LIN {X 0,Y 435.105,Z 1048.847,A -85,B 0,C 180,E1 20642.919,E2 20642.919} C_VEL
LIN {X 0,Y 432.049,Z 1065.311,A -85,B 0,C 180,E1 20641.068,E2 20641.068} C_VEL
LIN {X 0,Y 428.929,Z 1081.421,A -85,B 0,C 180,E1 20638.926,E2 20638.926} C_VEL
LIN {X 0,Y 426.223,Z 1095.243,A -85,B 0,C 180,E1 20636.769,E2 20636.769} C_VEL
LIN {X 0,Y 423.614,Z 1108.344,A -85,B 0,C 180,E1 20634.345,E2 20634.345} C_VEL
LIN {X 0,Y 421.322,Z 1120.264,A -85,B 0,C 180,E1 20631.728,E2 20631.728} C_VEL
LIN {X 0,Y 419.538,Z 1130.485,A -85,B 0,C 180,E1 20629.056,E2 20629.056} C_VEL
LIN {X 0,Y 418.131,Z 1139.349,A -85,B 0,C 180,E1 20626.246,E2 20626.246} C_VEL
LIN {X 0,Y 417.148,Z 1146.8,A -85,B 0,C 180,E1 20623.303,E2 20623.303} C_VEL
LIN {X 0,Y 416.528,Z 1152.908,A -85,B 0,C 180,E1 20620.201,E2 20620.201} C_VEL
LIN {X 0,Y 416.233,Z 1157.103,A -85,B 0,C 180,E1 20617.314,E2 20617.314} C_VEL
LIN {X 0,Y 416.088,Z 1159.912,A -85,B 0,C 180,E1 20614.272,E2 20614.272} C_VEL
LIN {X 0,Y 416.05,Z 1161.297,A -85,B 0,C 180,E1 20611.102,E2 20611.102} C_VEL
LIN {X 0,Y 416.047,Z 1161.219,A -85,B 0,C 180,E1 20608.21,E2 20608.21} C_VEL
LIN {X 0,Y 416.098,Z 1159.578,A -85,B 0,C 180,E1 20605.176,E2 20605.176} C_VEL
LIN {X 0,Y 416.291,Z 1156.297,A -85,B 0,C 180,E1 20601.993,E2 20601.993} C_VEL
LIN {X 0,Y 416.638,Z 1151.851,A -85,B 0,C 180,E1 20599.072,E2 20599.072} C_VEL
LIN {X 0,Y 417.28,Z 1145.733,A -85,B 0,C 180,E1 20596.137,E2 20596.137} C_VEL
LIN {X 0,Y 418.332,Z 1137.948,A -85,B 0,C 180,E1 20593.19,E2 20593.19} C_VEL
LIN {X 0,Y 419.837,Z 1128.815,A -85,B 0,C 180,E1 20590.38,E2 20590.38} C_VEL
LIN {X 0,Y 421.711,Z 1118.284,A -85,B 0,C 180,E1 20587.707,E2 20587.707} C_VEL
LIN {X 0,Y 423.979,Z 1106.39,A -85,B 0,C 180,E1 20585.181,E2 20585.181} C_VEL
LIN {X 0,Y 426.622,Z 1093.222,A -85,B 0,C 180,E1 20582.806,E2 20582.806} C_VEL
LIN {X 0,Y 429.496,Z 1078.65,A -85,B 0,C 180,E1 20580.581,E2 20580.581} C_VEL
LIN {X 0,Y 432.519,Z 1062.81,A -85,B 0,C 180,E1 20578.542,E2 20578.542} C_VEL
LIN {X 0,Y 435.66,Z 1045.506,A -85,B 0,C 180,E1 20576.657,E2 20576.657} C_VEL
LIN {X 0,Y 438.639,Z 1027.657,A -85,B 0,C 180,E1 20575.022,E2 20575.022} C_VEL
LIN {X 0,Y 441.258,Z 1009.727,A -85,B 0,C 180,E1 20573.664,E2 20573.664} C_VEL
LIN {X 0,Y 443.774,Z 989.808,A -85,B 0,C 180,E1 20572.414,E2 20572.414} C_VEL
LIN {X 0,Y 445.795,Z 970.199,A -85,B 0,C 180,E1 20571.428,E2 20571.428} C_VEL
LIN {X 0,Y 447.419,Z 949.171,A -85,B 0,C 180,E1 20570.621,E2 20570.621} C_VEL
LIN {X 0,Y 448.598,Z 926.606,A -85,B 0,C 180,E1 20570.002,E2 20570.002} C_VEL
LIN {X 0,Y 454.402,Z 736.319,A -85,B 0,C 180,E1 20566.605,E2 20566.605} C_VEL
LIN {X 0,Y 442.027,Z 717.492,A -85,B 0,C 180,E1 20564.566,E2 20564.566} C_VEL
LIN {X 0,Y 431.685,Z 703.053,A -85,B 0,C 180,E1 20562.738,E2 20562.738} C_VEL
LIN {X 0,Y 428.164,Z 698.288,A -85,B 0,C 180,E1 20562.083,E2 20562.083} C_VEL
LIN {X 0,Y 424.696,Z 693.577,A -85,B 0,C 180,E1 20561.419,E2 20561.419} C_VEL
LIN {X 0,Y 421.91,Z 689.861,A -85,B 0,C 180,E1 20560.872,E2 20560.872} C_VEL
LIN {X 0,Y 421.003,Z 688.483,A -85,B 0,C 180,E1 20560.687,E2 20560.687} C_VEL
LIN {X 0,Y 418.41,Z 685.788,A -85,B 0,C 180,E1 20560.182,E2 20560.182} C_VEL
LIN {X 0,Y 417.461,Z 683.308,A -85,B 0,C 180,E1 20559.856,E2 20559.856} C_VEL
LIN {X 0,Y 417.38,Z 682.765,A -85,B 0,C 180,E1 20559.525,E2 20559.525} C_VEL
LIN {X 0,Y 417.364,Z 682.695,A -85,B 0,C 180,E1 20555.602,E2 20555.602} C_VEL
LIN {X 0,Y 417.373,Z 682.695,A -85,B 0,C 180,E1 20551.805,E2 20551.805} C_VEL
LIN {X 0,Y 417.368,Z 682.712,A -85,B 0,C 180,E1 20547.876,E2 20547.876} C_VEL
LIN {X 0,Y 417.373,Z 682.728,A -85,B 0,C 180,E1 20544.033,E2 20544.033} C_VEL
LIN {X 0,Y 417.382,Z 682.725,A -85,B 0,C 180,E1 20540.18,E2 20540.18} C_VEL
LIN {X 0,Y 417.381,Z 682.726,A -85,B 0,C 180,E1 20536.277,E2 20536.277} C_VEL
LIN {X 0,Y 417.378,Z 682.734,A -85,B 0,C 180,E1 20532.451,E2 20532.451} C_VEL
LIN {X 0,Y 417.371,Z 682.744,A -85,B 0,C 180,E1 20528.542,E2 20528.542} C_VEL
LIN {X 0,Y 417.374,Z 682.745,A -85,B 0,C 180,E1 20524.672,E2 20524.672} C_VEL
LIN {X 0,Y 417.375,Z 682.733,A -85,B 0,C 180,E1 20520.824,E2 20520.824} C_VEL
LIN {X 0,Y 417.375,Z 682.725,A -85,B 0,C 180,E1 20516.979,E2 20516.979} C_VEL
LIN {X 0,Y 417.378,Z 682.728,A -85,B 0,C 180,E1 20513.121,E2 20513.121} C_VEL
LIN {X 0,Y 417.369,Z 682.736,A -85,B 0,C 180,E1 20509.165,E2 20509.165} C_VEL
LIN {X 0,Y 417.375,Z 682.723,A -85,B 0,C 180,E1 20505.29,E2 20505.29} C_VEL
LIN {X 0,Y 417.369,Z 682.707,A -85,B 0,C 180,E1 20501.421,E2 20501.421} C_VEL
LIN {X 0,Y 417.371,Z 682.743,A -85,B 0,C 180,E1 20497.611,E2 20497.611} C_VEL
LIN {X 0,Y 417.373,Z 682.731,A -85,B 0,C 180,E1 20493.693,E2 20493.693} C_VEL
LIN {X 0,Y 417.367,Z 682.716,A -85,B 0,C 180,E1 20489.796,E2 20489.796} C_VEL
LIN {X 0,Y 417.397,Z 682.931,A -85,B 0,C 180,E1 20486.613,E2 20486.613} C_VEL
LIN {X 0,Y 418.867,Z 686.47,A -85,B 0,C 180,E1 20485.878,E2 20485.878} C_VEL
LIN {X 0,Y 420.281,Z 689.046,A -85,B 0,C 180,E1 20485.349,E2 20485.349} C_VEL
LIN {X 0,Y 424.942,Z 697.897,A -85,B 0,C 180,E1 20483.635,E2 20483.635} C_VEL
LIN {X 0,Y 431.28,Z 710.634,A -85,B 0,C 180,E1 20481.376,E2 20481.376} C_VEL
LIN {X 0,Y 438.741,Z 726.744,A -85,B 0,C 180,E1 20478.806,E2 20478.806} C_VEL
LIN {X 0,Y 443.748,Z 738.403,A -85,B 0,C 180,E1 20477.164,E2 20477.164} C_VEL
LIN {X 0,Y 448.342,Z 747.008,A -85,B 0,C 180,E1 20476.364,E2 20476.364} C_VEL
LIN {X 0,Y 454.393,Z 794.703,A -85,B 0,C 180,E1 20474.578,E2 20474.578} C_VEL
LIN {X 0,Y 447.858,Z 1022.653,A -85,B 0,C 180,E1 20470.573,E2 20470.573} C_VEL
LIN {X 0,Y 446.684,Z 1054.914,A -85,B 0,C 180,E1 20469.961,E2 20469.961} C_VEL
LIN {X 0,Y 444.937,Z 1076.85,A -85,B 0,C 180,E1 20469.36,E2 20469.36} C_VEL
LIN {X 0,Y 442.616,Z 1098.688,A -85,B 0,C 180,E1 20468.528,E2 20468.528} C_VEL
LIN {X 0,Y 439.968,Z 1120.596,A -85,B 0,C 180,E1 20467.437,E2 20467.437} C_VEL
LIN {X 0,Y 437.183,Z 1141.229,A -85,B 0,C 180,E1 20466.16,E2 20466.16} C_VEL
LIN {X 0,Y 434.116,Z 1161.603,A -85,B 0,C 180,E1 20464.612,E2 20464.612} C_VEL
LIN {X 0,Y 431.045,Z 1181.633,A -85,B 0,C 180,E1 20462.791,E2 20462.791} C_VEL
LIN {X 0,Y 428.169,Z 1199.938,A -85,B 0,C 180,E1 20460.834,E2 20460.834} C_VEL
LIN {X 0,Y 425.46,Z 1217.379,A -85,B 0,C 180,E1 20458.646,E2 20458.646} C_VEL
LIN {X 0,Y 423.143,Z 1232.905,A -85,B 0,C 180,E1 20456.373,E2 20456.373} C_VEL
LIN {X 0,Y 421.041,Z 1248.049,A -85,B 0,C 180,E1 20453.809,E2 20453.809} C_VEL
LIN {X 0,Y 419.33,Z 1261.714,A -85,B 0,C 180,E1 20451.102,E2 20451.102} C_VEL
LIN {X 0,Y 418.06,Z 1273.181,A -85,B 0,C 180,E1 20448.402,E2 20448.402} C_VEL
LIN {X 0,Y 417.113,Z 1283.79,A -85,B 0,C 180,E1 20445.43,E2 20445.43} C_VEL
LIN {X 0,Y 416.542,Z 1292.034,A -85,B 0,C 180,E1 20442.617,E2 20442.617} C_VEL
LIN {X 0,Y 416.215,Z 1298.402,A -85,B 0,C 180,E1 20439.82,E2 20439.82} C_VEL
LIN {X 0,Y 416.067,Z 1303.414,A -85,B 0,C 180,E1 20436.901,E2 20436.901} C_VEL
LIN {X 0,Y 416.007,Z 1306.377,A -85,B 0,C 180,E1 20434.273,E2 20434.273} C_VEL
LIN {X 0,Y 415.991,Z 1308.055,A -85,B 0,C 180,E1 20431.377,E2 20431.377} C_VEL
LIN {X 0,Y 415.995,Z 1308.108,A -85,B 0,C 180,E1 20428.898,E2 20428.898} C_VEL
LIN {X 0,Y 415.999,Z 1306.625,A -85,B 0,C 180,E1 20426.003,E2 20426.003} C_VEL
LIN {X 0,Y 416.055,Z 1303.768,A -85,B 0,C 180,E1 20423.376,E2 20423.376} C_VEL
LIN {X 0,Y 416.191,Z 1298.965,A -85,B 0,C 180,E1 20420.459,E2 20420.459} C_VEL
LIN {X 0,Y 416.502,Z 1292.812,A -85,B 0,C 180,E1 20417.699,E2 20417.699} C_VEL
LIN {X 0,Y 417.043,Z 1284.682,A -85,B 0,C 180,E1 20414.852,E2 20414.852} C_VEL
LIN {X 0,Y 417.901,Z 1274.869,A -85,B 0,C 180,E1 20412.023,E2 20412.023} C_VEL
LIN {X 0,Y 419.1,Z 1263.623,A -85,B 0,C 180,E1 20409.324,E2 20409.324} C_VEL
LIN {X 0,Y 420.728,Z 1250.326,A -85,B 0,C 180,E1 20406.618,E2 20406.618} C_VEL
LIN {X 0,Y 422.75,Z 1235.627,A -85,B 0,C 180,E1 20404.053,E2 20404.053} C_VEL
LIN {X 0,Y 425.143,Z 1219.477,A -85,B 0,C 180,E1 20401.637,E2 20401.637} C_VEL
LIN {X 0,Y 427.804,Z 1202.297,A -85,B 0,C 180,E1 20399.448,E2 20399.448} C_VEL
LIN {X 0,Y 430.827,Z 1183.015,A -85,B 0,C 180,E1 20397.346,E2 20397.346} C_VEL
LIN {X 0,Y 433.727,Z 1164.363,A -85,B 0,C 180,E1 20395.613,E2 20395.613} C_VEL
LIN {X 0,Y 436.693,Z 1144.354,A -85,B 0,C 180,E1 20394.064,E2 20394.064} C_VEL
LIN {X 0,Y 439.511,Z 1124.075,A -85,B 0,C 180,E1 20392.763,E2 20392.763} C_VEL
LIN {X 0,Y 442.136,Z 1103.214,A -85,B 0,C 180,E1 20391.671,E2 20391.671} C_VEL
LIN {X 0,Y 444.459,Z 1081.387,A -85,B 0,C 180,E1 20390.793,E2 20390.793} C_VEL
LIN {X 0,Y 446.394,Z 1058.963,A -85,B 0,C 180,E1 20390.139,E2 20390.139} C_VEL
LIN {X 0,Y 447.524,Z 1034.567,A -85,B 0,C 180,E1 20389.636,E2 20389.636} C_VEL
LIN {X 0,Y 453.824,Z 812.838,A -85,B 0,C 180,E1 20385.744,E2 20385.744} C_VEL
LIN {X 0,Y 454.249,Z 792.558,A -85,B 0,C 180,E1 20385.364,E2 20385.364} C_VEL
LIN {X 0,Y 448.083,Z 746.171,A -85,B 0,C 180,E1 20383.591,E2 20383.591} C_VEL
LIN {X 0,Y 443.103,Z 737.098,A -85,B 0,C 180,E1 20382.693,E2 20382.693} C_VEL
LIN {X 0,Y 435.309,Z 719.135,A -85,B 0,C 180,E1 20380.025,E2 20380.025} C_VEL
LIN {X 0,Y 427.831,Z 703.608,A -85,B 0,C 180,E1 20377.418,E2 20377.418} C_VEL
LIN {X 0,Y 421.698,Z 691.586,A -85,B 0,C 180,E1 20375.181,E2 20375.181} C_VEL
LIN {X 0,Y 419.231,Z 686.954,A -85,B 0,C 180,E1 20374.253,E2 20374.253} C_VEL
LIN {X 0,Y 417.47,Z 683.338,A -85,B 0,C 180,E1 20373.508,E2 20373.508} C_VEL
LIN {X 0,Y 417.376,Z 682.76,A -85,B 0,C 180,E1 20373.106,E2 20373.106} C_VEL
LIN {X 0,Y 417.368,Z 682.713,A -85,B 0,C 180,E1 20369.255,E2 20369.255} C_VEL
LIN {X 0,Y 417.373,Z 682.714,A -85,B 0,C 180,E1 20365.392,E2 20365.392} C_VEL
LIN {X 0,Y 417.371,Z 682.743,A -85,B 0,C 180,E1 20361.501,E2 20361.501} C_VEL
LIN {X 0,Y 417.371,Z 682.724,A -85,B 0,C 180,E1 20357.556,E2 20357.556} C_VEL
LIN {X 0,Y 417.369,Z 682.706,A -85,B 0,C 180,E1 20353.719,E2 20353.719} C_VEL
LIN {X 0,Y 417.37,Z 682.747,A -85,B 0,C 180,E1 20349.793,E2 20349.793} C_VEL
LIN {X 0,Y 417.377,Z 682.74,A -85,B 0,C 180,E1 20345.912,E2 20345.912} C_VEL
LIN {X 0,Y 417.368,Z 682.729,A -85,B 0,C 180,E1 20342.059,E2 20342.059} C_VEL
LIN {X 0,Y 417.373,Z 682.723,A -85,B 0,C 180,E1 20338.215,E2 20338.215} C_VEL
LIN {X 0,Y 417.382,Z 682.73,A -85,B 0,C 180,E1 20334.363,E2 20334.363} C_VEL
LIN {X 0,Y 417.379,Z 682.744,A -85,B 0,C 180,E1 20330.485,E2 20330.485} C_VEL
LIN {X 0,Y 417.379,Z 682.743,A -85,B 0,C 180,E1 20326.549,E2 20326.549} C_VEL
LIN {X 0,Y 417.37,Z 682.739,A -85,B 0,C 180,E1 20322.719,E2 20322.719} C_VEL
LIN {X 0,Y 417.376,Z 682.732,A -85,B 0,C 180,E1 20318.793,E2 20318.793} C_VEL
LIN {X 0,Y 417.379,Z 682.729,A -85,B 0,C 180,E1 20314.89,E2 20314.89} C_VEL
LIN {X 0,Y 417.375,Z 682.682,A -85,B 0,C 180,E1 20310.97,E2 20310.97} C_VEL
LIN {X 0,Y 417.379,Z 682.731,A -85,B 0,C 180,E1 20307.058,E2 20307.058} C_VEL
LIN {X 0,Y 417.365,Z 682.682,A -85,B 0,C 180,E1 20303.142,E2 20303.142} C_VEL
LIN {X 0,Y 417.407,Z 683.001,A -85,B 0,C 180,E1 20300.138,E2 20300.138} C_VEL
LIN {X 0,Y 417.795,Z 684.484,A -85,B 0,C 180,E1 20299.859,E2 20299.859} C_VEL
LIN {X 0,Y 419.777,Z 687.508,A -85,B 0,C 180,E1 20299.439,E2 20299.439} C_VEL
LIN {X 0,Y 421.602,Z 689.242,A -85,B 0,C 180,E1 20299.091,E2 20299.091} C_VEL
LIN {X 0,Y 424.212,Z 693.11,A -85,B 0,C 180,E1 20298.568,E2 20298.568} C_VEL
LIN {X 0,Y 425.888,Z 695.117,A -85,B 0,C 180,E1 20298.251,E2 20298.251} C_VEL
LIN {X 0,Y 436.949,Z 710.273,A -85,B 0,C 180,E1 20296.218,E2 20296.218} C_VEL
LIN {X 0,Y 448.56,Z 727.22,A -85,B 0,C 180,E1 20294.243,E2 20294.243} C_VEL
LIN {X 0,Y 454.437,Z 736.746,A -85,B 0,C 180,E1 20293.287,E2 20293.287} C_VEL
LIN {X 0,Y 448.516,Z 928.762,A -85,B 0,C 180,E1 20289.861,E2 20289.861} C_VEL
LIN {X 0,Y 447.322,Z 950.387,A -85,B 0,C 180,E1 20289.248,E2 20289.248} C_VEL
LIN {X 0,Y 445.662,Z 971.471,A -85,B 0,C 180,E1 20288.421,E2 20288.421} C_VEL
LIN {X 0,Y 443.727,Z 990.201,A -85,B 0,C 180,E1 20287.472,E2 20287.472} C_VEL
LIN {X 0,Y 441.269,Z 1009.589,A -85,B 0,C 180,E1 20286.255,E2 20286.255} C_VEL
LIN {X 0,Y 438.656,Z 1027.541,A -85,B 0,C 180,E1 20284.897,E2 20284.897} C_VEL
LIN {X 0,Y 438.08,Z 1030.915,A -85,B 0,C 180,E1 20284.604,E2 20284.604} C_VEL
LIN {X 0,Y 436.23,Z 1037.563,A -85,B 0,C 180,E1 20284.109,E2 20284.109} C_VEL
LIN {X 0,Y 428.568,Z 1054.082,A -85,B 0,C 180,E1 20283.003,E2 20283.003} C_VEL
LIN {X 0,Y 426.613,Z 1060.13,A -85,B 0,C 180,E1 20282.411,E2 20282.411} C_VEL
LIN {X 0,Y 423.452,Z 1075.881,A -85,B 0,C 180,E1 20280.429,E2 20280.429} C_VEL
LIN {X 0,Y 420.375,Z 1090.636,A -85,B 0,C 180,E1 20278.249,E2 20278.249} C_VEL
LIN {X 0,Y 417.495,Z 1104.49,A -85,B 0,C 180,E1 20275.84,E2 20275.84} C_VEL
LIN {X 0,Y 414.929,Z 1116.824,A -85,B 0,C 180,E1 20273.277,E2 20273.277} C_VEL
LIN {X 0,Y 412.756,Z 1127.792,A -85,B 0,C 180,E1 20270.563,E2 20270.563} C_VEL
LIN {X 0,Y 411.036,Z 1137.421,A -85,B 0,C 180,E1 20267.701,E2 20267.701} C_VEL
LIN {X 0,Y 409.795,Z 1145.607,A -85,B 0,C 180,E1 20264.699,E2 20264.699} C_VEL
LIN {X 0,Y 408.965,Z 1151.989,A -85,B 0,C 180,E1 20261.708,E2 20261.708} C_VEL
LIN {X 0,Y 408.487,Z 1157.208,A -85,B 0,C 180,E1 20258.445,E2 20258.445} C_VEL
LIN {X 0,Y 408.267,Z 1160.504,A -85,B 0,C 180,E1 20255.481,E2 20255.481} C_VEL
LIN {X 0,Y 408.177,Z 1162.284,A -85,B 0,C 180,E1 20252.527,E2 20252.527} C_VEL
LIN {X 0,Y 408.163,Z 1162.783,A -85,B 0,C 180,E1 20249.439,E2 20249.439} C_VEL
LIN {X 0,Y 408.198,Z 1161.908,A -85,B 0,C 180,E1 20246.489,E2 20246.489} C_VEL
LIN {X 0,Y 408.326,Z 1159.468,A -85,B 0,C 180,E1 20243.392,E2 20243.392} C_VEL
LIN {X 0,Y 408.629,Z 1155.534,A -85,B 0,C 180,E1 20240.28,E2 20240.28} C_VEL
LIN {X 0,Y 409.213,Z 1149.988,A -85,B 0,C 180,E1 20237.154,E2 20237.154} C_VEL
LIN {X 0,Y 410.165,Z 1142.911,A -85,B 0,C 180,E1 20234.156,E2 20234.156} C_VEL
LIN {X 0,Y 411.614,Z 1134.066,A -85,B 0,C 180,E1 20231.152,E2 20231.152} C_VEL
LIN {X 0,Y 413.436,Z 1124.367,A -85,B 0,C 180,E1 20228.433,E2 20228.433} C_VEL
LIN {X 0,Y 415.78,Z 1112.678,A -85,B 0,C 180,E1 20225.719,E2 20225.719} C_VEL
LIN {X 0,Y 418.345,Z 1100.279,A -85,B 0,C 180,E1 20223.3,E2 20223.3} C_VEL
LIN {X 0,Y 421.323,Z 1086.246,A -85,B 0,C 180,E1 20220.968,E2 20220.968} C_VEL
LIN {X 0,Y 424.402,Z 1071.251,A -85,B 0,C 180,E1 20218.862,E2 20218.862} C_VEL
LIN {X 0,Y 427.599,Z 1054.8,A -85,B 0,C 180,E1 20216.908,E2 20216.908} C_VEL
LIN {X 0,Y 430.875,Z 1036.819,A -85,B 0,C 180,E1 20215.111,E2 20215.111} C_VEL
LIN {X 0,Y 433.817,Z 1018.714,A -85,B 0,C 180,E1 20213.597,E2 20213.597} C_VEL
LIN {X 0,Y 436.474,Z 999.731,A -85,B 0,C 180,E1 20212.294,E2 20212.294} C_VEL
LIN {X 0,Y 438.82,Z 980.059,A -85,B 0,C 180,E1 20211.193,E2 20211.193} C_VEL
LIN {X 0,Y 440.62,Z 960.698,A -85,B 0,C 180,E1 20210.337,E2 20210.337} C_VEL
LIN {X 0,Y 442.044,Z 939.071,A -85,B 0,C 180,E1 20209.62,E2 20209.62} C_VEL
LIN {X 0,Y 442.941,Z 916.712,A -85,B 0,C 180,E1 20209.113,E2 20209.113} C_VEL
LIN {X 0,Y 448.627,Z 739.883,A -85,B 0,C 180,E1 20205.952,E2 20205.952} C_VEL
LIN {X 0,Y 436.717,Z 721.804,A -85,B 0,C 180,E1 20203.925,E2 20203.925} C_VEL
LIN {X 0,Y 424.925,Z 705.191,A -85,B 0,C 180,E1 20201.752,E2 20201.752} C_VEL
LIN {X 0,Y 420.465,Z 699.412,A -85,B 0,C 180,E1 20200.885,E2 20200.885} C_VEL
LIN {X 0,Y 417.089,Z 694.834,A -85,B 0,C 180,E1 20200.2,E2 20200.2} C_VEL
LIN {X 0,Y 414.227,Z 691.212,A -85,B 0,C 180,E1 20199.609,E2 20199.609} C_VEL
LIN {X 0,Y 413.366,Z 689.664,A -85,B 0,C 180,E1 20199.416,E2 20199.416} C_VEL
LIN {X 0,Y 410.623,Z 687.015,A -85,B 0,C 180,E1 20198.852,E2 20198.852} C_VEL
LIN {X 0,Y 409.556,Z 684.409,A -85,B 0,C 180,E1 20198.502,E2 20198.502} C_VEL
LIN {X 0,Y 409.443,Z 683.75,A -85,B 0,C 180,E1 20198.158,E2 20198.158} C_VEL
LIN {X 0,Y 409.433,Z 683.723,A -85,B 0,C 180,E1 20194.172,E2 20194.172} C_VEL
LIN {X 0,Y 409.42,Z 683.66,A -85,B 0,C 180,E1 20190.204,E2 20190.204} C_VEL
LIN {X 0,Y 409.438,Z 683.734,A -85,B 0,C 180,E1 20186.338,E2 20186.338} C_VEL
LIN {X 0,Y 409.446,Z 683.733,A -85,B 0,C 180,E1 20182.393,E2 20182.393} C_VEL
LIN {X 0,Y 409.443,Z 683.73,A -85,B 0,C 180,E1 20178.51,E2 20178.51} C_VEL
LIN {X 0,Y 409.446,Z 683.726,A -85,B 0,C 180,E1 20174.568,E2 20174.568} C_VEL
LIN {X 0,Y 409.429,Z 683.717,A -85,B 0,C 180,E1 20170.696,E2 20170.696} C_VEL
LIN {X 0,Y 409.434,Z 683.71,A -85,B 0,C 180,E1 20166.732,E2 20166.732} C_VEL
LIN {X 0,Y 409.435,Z 683.715,A -85,B 0,C 180,E1 20162.8,E2 20162.8} C_VEL
LIN {X 0,Y 409.438,Z 683.728,A -85,B 0,C 180,E1 20158.881,E2 20158.881} C_VEL
LIN {X 0,Y 409.443,Z 683.734,A -85,B 0,C 180,E1 20154.957,E2 20154.957} C_VEL
LIN {X 0,Y 409.432,Z 683.727,A -85,B 0,C 180,E1 20151.15,E2 20151.15} C_VEL
LIN {X 0,Y 409.427,Z 683.69,A -85,B 0,C 180,E1 20147.16,E2 20147.16} C_VEL
LIN {X 0,Y 409.437,Z 683.732,A -85,B 0,C 180,E1 20143.252,E2 20143.252} C_VEL
LIN {X 0,Y 409.434,Z 683.711,A -85,B 0,C 180,E1 20139.262,E2 20139.262} C_VEL
LIN {X 0,Y 409.428,Z 683.698,A -85,B 0,C 180,E1 20135.289,E2 20135.289} C_VEL
LIN {X 0,Y 409.439,Z 683.706,A -85,B 0,C 180,E1 20131.404,E2 20131.404} C_VEL
LIN {X 0,Y 409.47,Z 683.98,A -85,B 0,C 180,E1 20127.88,E2 20127.88} C_VEL
LIN {X 0,Y 410.92,Z 687.453,A -85,B 0,C 180,E1 20127.139,E2 20127.139} C_VEL
LIN {X 0,Y 412.041,Z 689.096,A -85,B 0,C 180,E1 20126.742,E2 20126.742} C_VEL
LIN {X 0,Y 419.283,Z 703.09,A -85,B 0,C 180,E1 20123.938,E2 20123.938} C_VEL
LIN {X 0,Y 426.639,Z 718.002,A -85,B 0,C 180,E1 20121.264,E2 20121.264} C_VEL
LIN {X 0,Y 434.494,Z 735.565,A -85,B 0,C 180,E1 20118.513,E2 20118.513} C_VEL
LIN {X 0,Y 442.987,Z 750.989,A -85,B 0,C 180,E1 20116.973,E2 20116.973} C_VEL
LIN {X 0,Y 448.544,Z 796.227,A -85,B 0,C 180,E1 20115.254,E2 20115.254} C_VEL
LIN {X 0,Y 441.664,Z 1023.492,A -85,B 0,C 180,E1 20111.217,E2 20111.217} C_VEL
LIN {X 0,Y 440.442,Z 1054.316,A -85,B 0,C 180,E1 20110.618,E2 20110.618} C_VEL
LIN {X 0,Y 438.561,Z 1076.754,A -85,B 0,C 180,E1 20109.993,E2 20109.993} C_VEL
LIN {X 0,Y 436.152,Z 1098.005,A -85,B 0,C 180,E1 20109.165,E2 20109.165} C_VEL
LIN {X 0,Y 433.272,Z 1120.306,A -85,B 0,C 180,E1 20108.034,E2 20108.034} C_VEL
LIN {X 0,Y 430.336,Z 1140.811,A -85,B 0,C 180,E1 20106.738,E2 20106.738} C_VEL
LIN {X 0,Y 427.232,Z 1160.274,A -85,B 0,C 180,E1 20105.238,E2 20105.238} C_VEL
LIN {X 0,Y 423.999,Z 1180.146,A -85,B 0,C 180,E1 20103.407,E2 20103.407} C_VEL
LIN {X 0,Y 420.938,Z 1198.448,A -85,B 0,C 180,E1 20101.424,E2 20101.424} C_VEL
LIN {X 0,Y 418.074,Z 1215.894,A -85,B 0,C 180,E1 20099.2,E2 20099.2} C_VEL
LIN {X 0,Y 415.484,Z 1232.153,A -85,B 0,C 180,E1 20096.772,E2 20096.772} C_VEL
LIN {X 0,Y 413.14,Z 1248.081,A -85,B 0,C 180,E1 20093.99,E2 20093.99} C_VEL
LIN {X 0,Y 411.377,Z 1261.519,A -85,B 0,C 180,E1 20091.231,E2 20091.231} C_VEL
LIN {X 0,Y 410.081,Z 1272.853,A -85,B 0,C 180,E1 20088.476,E2 20088.476} C_VEL
LIN {X 0,Y 409.164,Z 1282.788,A -85,B 0,C 180,E1 20085.593,E2 20085.593} C_VEL
LIN {X 0,Y 408.595,Z 1290.954,A -85,B 0,C 180,E1 20082.722,E2 20082.722} C_VEL
LIN {X 0,Y 408.285,Z 1297.267,A -85,B 0,C 180,E1 20079.87,E2 20079.87} C_VEL
LIN {X 0,Y 408.159,Z 1302.189,A -85,B 0,C 180,E1 20076.894,E2 20076.894} C_VEL
LIN {X 0,Y 408.115,Z 1305.107,A -85,B 0,C 180,E1 20074.215,E2 20074.215} C_VEL
LIN {X 0,Y 408.113,Z 1306.691,A -85,B 0,C 180,E1 20071.263,E2 20071.263} C_VEL
LIN {X 0,Y 408.113,Z 1306.69,A -85,B 0,C 180,E1 20068.737,E2 20068.737} C_VEL
LIN {X 0,Y 408.115,Z 1305.104,A -85,B 0,C 180,E1 20065.785,E2 20065.785} C_VEL
LIN {X 0,Y 408.159,Z 1302.184,A -85,B 0,C 180,E1 20063.106,E2 20063.106} C_VEL
LIN {X 0,Y 408.285,Z 1297.266,A -85,B 0,C 180,E1 20060.13,E2 20060.13} C_VEL
LIN {X 0,Y 408.595,Z 1290.956,A -85,B 0,C 180,E1 20057.278,E2 20057.278} C_VEL
LIN {X 0,Y 409.163,Z 1282.786,A -85,B 0,C 180,E1 20054.407,E2 20054.407} C_VEL
LIN {X 0,Y 410.081,Z 1272.844,A -85,B 0,C 180,E1 20051.521,E2 20051.521} C_VEL
LIN {X 0,Y 411.378,Z 1261.524,A -85,B 0,C 180,E1 20048.769,E2 20048.769} C_VEL
LIN {X 0,Y 413.14,Z 1248.086,A -85,B 0,C 180,E1 20046.01,E2 20046.01} C_VEL
LIN {X 0,Y 415.484,Z 1232.159,A -85,B 0,C 180,E1 20043.228,E2 20043.228} C_VEL
LIN {X 0,Y 418.074,Z 1215.897,A -85,B 0,C 180,E1 20040.8,E2 20040.8} C_VEL
LIN {X 0,Y 420.938,Z 1198.45,A -85,B 0,C 180,E1 20038.576,E2 20038.576} C_VEL
LIN {X 0,Y 424.002,Z 1180.139,A -85,B 0,C 180,E1 20036.593,E2 20036.593} C_VEL
LIN {X 0,Y 427.232,Z 1160.272,A -85,B 0,C 180,E1 20034.762,E2 20034.762} C_VEL
LIN {X 0,Y 430.334,Z 1140.804,A -85,B 0,C 180,E1 20033.262,E2 20033.262} C_VEL
LIN {X 0,Y 433.27,Z 1120.283,A -85,B 0,C 180,E1 20031.965,E2 20031.965} C_VEL
LIN {X 0,Y 436.15,Z 1097.977,A -85,B 0,C 180,E1 20030.835,E2 20030.835} C_VEL
LIN {X 0,Y 438.605,Z 1076.219,A -85,B 0,C 180,E1 20029.992,E2 20029.992} C_VEL
LIN {X 0,Y 440.462,Z 1053.904,A -85,B 0,C 180,E1 20029.374,E2 20029.374} C_VEL
LIN {X 0,Y 441.688,Z 1022.224,A -85,B 0,C 180,E1 20028.762,E2 20028.762} C_VEL
LIN {X 0,Y 448.557,Z 795.233,A -85,B 0,C 180,E1 20024.731,E2 20024.731} C_VEL
LIN {X 0,Y 442.801,Z 750.318,A -85,B 0,C 180,E1 20022.994,E2 20022.994} C_VEL
LIN {X 0,Y 434.069,Z 734.703,A -85,B 0,C 180,E1 20021.383,E2 20021.383} C_VEL
LIN {X 0,Y 426.377,Z 717.523,A -85,B 0,C 180,E1 20018.66,E2 20018.66} C_VEL
LIN {X 0,Y 418.608,Z 701.688,A -85,B 0,C 180,E1 20015.816,E2 20015.816} C_VEL
LIN {X 0,Y 413.66,Z 692.377,A -85,B 0,C 180,E1 20013.941,E2 20013.941} C_VEL
LIN {X 0,Y 411.273,Z 687.9,A -85,B 0,C 180,E1 20012.995,E2 20012.995} C_VEL
LIN {X 0,Y 409.553,Z 684.429,A -85,B 0,C 180,E1 20012.237,E2 20012.237} C_VEL
LIN {X 0,Y 409.45,Z 683.827,A -85,B 0,C 180,E1 20011.999,E2 20011.999} C_VEL
LIN {X 0,Y 409.43,Z 683.716,A -85,B 0,C 180,E1 20008.12,E2 20008.12} C_VEL
LIN {X 0,Y 409.433,Z 683.699,A -85,B 0,C 180,E1 20004.221,E2 20004.221} C_VEL
LIN {X 0,Y 409.429,Z 683.705,A -85,B 0,C 180,E1 20000.439,E2 20000.439} C_VEL
LIN {X 0,Y 409.435,Z 683.733,A -85,B 0,C 180,E1 19996.456,E2 19996.456} C_VEL
LIN {X 0,Y 409.431,Z 683.691,A -85,B 0,C 180,E1 19992.553,E2 19992.553} C_VEL
LIN {X 0,Y 409.43,Z 683.726,A -85,B 0,C 180,E1 19988.708,E2 19988.708} C_VEL
LIN {X 0,Y 409.439,Z 683.732,A -85,B 0,C 180,E1 19984.762,E2 19984.762} C_VEL
LIN {X 0,Y 409.445,Z 683.732,A -85,B 0,C 180,E1 19980.839,E2 19980.839} C_VEL
LIN {X 0,Y 409.436,Z 683.719,A -85,B 0,C 180,E1 19976.92,E2 19976.92} C_VEL
LIN {X 0,Y 409.442,Z 683.71,A -85,B 0,C 180,E1 19972.986,E2 19972.986} C_VEL
LIN {X 0,Y 409.43,Z 683.715,A -85,B 0,C 180,E1 19969.017,E2 19969.017} C_VEL
LIN {X 0,Y 409.433,Z 683.724,A -85,B 0,C 180,E1 19965.142,E2 19965.142} C_VEL
LIN {X 0,Y 409.442,Z 683.728,A -85,B 0,C 180,E1 19961.195,E2 19961.195} C_VEL
LIN {X 0,Y 409.445,Z 683.73,A -85,B 0,C 180,E1 19957.304,E2 19957.304} C_VEL
LIN {X 0,Y 409.442,Z 683.731,A -85,B 0,C 180,E1 19953.299,E2 19953.299} C_VEL
LIN {X 0,Y 409.43,Z 683.659,A -85,B 0,C 180,E1 19949.472,E2 19949.472} C_VEL
LIN {X 0,Y 409.431,Z 683.713,A -85,B 0,C 180,E1 19945.489,E2 19945.489} C_VEL
LIN {X 0,Y 409.451,Z 683.823,A -85,B 0,C 180,E1 19941.576,E2 19941.576} C_VEL
LIN {X 0,Y 409.789,Z 685.278,A -85,B 0,C 180,E1 19941.249,E2 19941.249} C_VEL
LIN {X 0,Y 411.735,Z 688.393,A -85,B 0,C 180,E1 19940.803,E2 19940.803} C_VEL
LIN {X 0,Y 413.726,Z 690.186,A -85,B 0,C 180,E1 19940.401,E2 19940.401} C_VEL
LIN {X 0,Y 416.322,Z 694.105,A -85,B 0,C 180,E1 19939.846,E2 19939.846} C_VEL
LIN {X 0,Y 418.085,Z 696.058,A -85,B 0,C 180,E1 19939.495,E2 19939.495} C_VEL
LIN {X 0,Y 421.446,Z 700.432,A -85,B 0,C 180,E1 19938.825,E2 19938.825} C_VEL
LIN {X 0,Y 433.471,Z 717.183,A -85,B 0,C 180,E1 19936.554,E2 19936.554} C_VEL
LIN {X 0,Y 444.369,Z 733.25,A -85,B 0,C 180,E1 19934.659,E2 19934.659} C_VEL
LIN {X 0,Y 448.638,Z 740.22,A -85,B 0,C 180,E1 19933.943,E2 19933.943} C_VEL
LIN {X 0,Y 442.482,Z 929.972,A -85,B 0,C 180,E1 19930.522,E2 19930.522} C_VEL
LIN {X 0,Y 441.248,Z 951.668,A -85,B 0,C 180,E1 19929.901,E2 19929.901} C_VEL
LIN {X 0,Y 439.517,Z 972.872,A -85,B 0,C 180,E1 19929.06,E2 19929.06} C_VEL
LIN {X 0,Y 437.502,Z 991.601,A -85,B 0,C 180,E1 19928.1,E2 19928.1} C_VEL
LIN {X 0,Y 434.941,Z 1010.986,A -85,B 0,C 180,E1 19926.868,E2 19926.868} C_VEL
LIN {X 0,Y 432.166,Z 1029.193,A -85,B 0,C 180,E1 19925.473,E2 19925.473} C_VEL
LIN {X 0,Y 429.088,Z 1046.793,A -85,B 0,C 180,E1 19923.842,E2 19923.842} C_VEL
LIN {X 0,Y 426.613,Z 1060.13,A -85,B 0,C 180,E1 19922.411,E2 19922.411} C_VEL
LIN {X 0,Y 424.627,Z 1066.077,A -85,B 0,C 180,E1 19921.787,E2 19921.787} C_VEL
LIN {X 0,Y 416.591,Z 1081.252,A -85,B 0,C 180,E1 19920.339,E2 19920.339} C_VEL
LIN {X 0,Y 414.612,Z 1086.579,A -85,B 0,C 180,E1 19919.633,E2 19919.633} C_VEL
LIN {X 0,Y 411.358,Z 1101.213,A -85,B 0,C 180,E1 19917.19,E2 19917.19} C_VEL
LIN {X 0,Y 408.473,Z 1114.342,A -85,B 0,C 180,E1 19914.589,E2 19914.589} C_VEL
LIN {X 0,Y 405.987,Z 1126.003,A -85,B 0,C 180,E1 19911.831,E2 19911.831} C_VEL
LIN {X 0,Y 404.023,Z 1135.768,A -85,B 0,C 180,E1 19909.028,E2 19909.028} C_VEL
LIN {X 0,Y 402.421,Z 1144.817,A -85,B 0,C 180,E1 19905.861,E2 19905.861} C_VEL
LIN {X 0,Y 401.407,Z 1151.767,A -85,B 0,C 180,E1 19902.808,E2 19902.808} C_VEL
LIN {X 0,Y 400.81,Z 1157.016,A -85,B 0,C 180,E1 19899.766,E2 19899.766} C_VEL
LIN {X 0,Y 400.469,Z 1160.912,A -85,B 0,C 180,E1 19896.595,E2 19896.595} C_VEL
LIN {X 0,Y 400.321,Z 1163.319,A -85,B 0,C 180,E1 19893.436,E2 19893.436} C_VEL
LIN {X 0,Y 400.284,Z 1164.181,A -85,B 0,C 180,E1 19890.429,E2 19890.429} C_VEL
LIN {X 0,Y 400.305,Z 1163.655,A -85,B 0,C 180,E1 19887.28,E2 19887.28} C_VEL
LIN {X 0,Y 400.419,Z 1161.854,A -85,B 0,C 180,E1 19884.268,E2 19884.268} C_VEL
LIN {X 0,Y 400.686,Z 1158.356,A -85,B 0,C 180,E1 19881.1,E2 19881.1} C_VEL
LIN {X 0,Y 401.205,Z 1153.29,A -85,B 0,C 180,E1 19877.917,E2 19877.917} C_VEL
LIN {X 0,Y 402.129,Z 1146.875,A -85,B 0,C 180,E1 19874.867,E2 19874.867} C_VEL
LIN {X 0,Y 403.491,Z 1138.669,A -85,B 0,C 180,E1 19871.807,E2 19871.807} C_VEL
LIN {X 0,Y 405.35,Z 1128.992,A -85,B 0,C 180,E1 19868.892,E2 19868.892} C_VEL
LIN {X 0,Y 407.816,Z 1117.323,A -85,B 0,C 180,E1 19865.985,E2 19865.985} C_VEL
LIN {X 0,Y 410.594,Z 1104.833,A -85,B 0,C 180,E1 19863.381,E2 19863.381} C_VEL
LIN {X 0,Y 413.689,Z 1090.811,A -85,B 0,C 180,E1 19860.936,E2 19860.936} C_VEL
LIN {X 0,Y 416.961,Z 1075.792,A -85,B 0,C 180,E1 19858.725,E2 19858.725} C_VEL
LIN {X 0,Y 420.255,Z 1060.005,A -85,B 0,C 180,E1 19856.744,E2 19856.744} C_VEL
LIN {X 0,Y 423.614,Z 1042.666,A -85,B 0,C 180,E1 19854.92,E2 19854.92} C_VEL
LIN {X 0,Y 426.778,Z 1024.426,A -85,B 0,C 180,E1 19853.316,E2 19853.316} C_VEL
LIN {X 0,Y 429.683,Z 1005.489,A -85,B 0,C 180,E1 19851.93,E2 19851.93} C_VEL
LIN {X 0,Y 432.066,Z 986.893,A -85,B 0,C 180,E1 19850.821,E2 19850.821} C_VEL
LIN {X 0,Y 434.212,Z 966.003,A -85,B 0,C 180,E1 19849.833,E2 19849.833} C_VEL
LIN {X 0,Y 435.836,Z 945.016,A -85,B 0,C 180,E1 19849.079,E2 19849.079} C_VEL
LIN {X 0,Y 436.764,Z 924.703,A -85,B 0,C 180,E1 19848.567,E2 19848.567} C_VEL
LIN {X 0,Y 442.819,Z 743.347,A -85,B 0,C 180,E1 19845.268,E2 19845.268} C_VEL
LIN {X 0,Y 431.01,Z 725.383,A -85,B 0,C 180,E1 19843.184,E2 19843.184} C_VEL
LIN {X 0,Y 420.536,Z 710.749,A -85,B 0,C 180,E1 19841.193,E2 19841.193} C_VEL
LIN {X 0,Y 413.22,Z 701.036,A -85,B 0,C 180,E1 19839.702,E2 19839.702} C_VEL
LIN {X 0,Y 409.384,Z 695.98,A -85,B 0,C 180,E1 19838.88,E2 19838.88} C_VEL
LIN {X 0,Y 406.535,Z 692.467,A -85,B 0,C 180,E1 19838.256,E2 19838.256} C_VEL
LIN {X 0,Y 405.366,Z 690.586,A -85,B 0,C 180,E1 19837.982,E2 19837.982} C_VEL
LIN {X 0,Y 402.656,Z 687.932,A -85,B 0,C 180,E1 19837.384,E2 19837.384} C_VEL
LIN {X 0,Y 401.598,Z 685.305,A -85,B 0,C 180,E1 19836.995,E2 19836.995} C_VEL
LIN {X 0,Y 401.488,Z 684.682,A -85,B 0,C 180,E1 19836.527,E2 19836.527} C_VEL
LIN {X 0,Y 401.491,Z 684.689,A -85,B 0,C 180,E1 19832.542,E2 19832.542} C_VEL
LIN {X 0,Y 401.499,Z 684.661,A -85,B 0,C 180,E1 19828.564,E2 19828.564} C_VEL
LIN {X 0,Y 401.502,Z 684.702,A -85,B 0,C 180,E1 19824.575,E2 19824.575} C_VEL
LIN {X 0,Y 401.504,Z 684.702,A -85,B 0,C 180,E1 19820.709,E2 19820.709} C_VEL
LIN {X 0,Y 401.5,Z 684.706,A -85,B 0,C 180,E1 19816.791,E2 19816.791} C_VEL
LIN {X 0,Y 401.492,Z 684.72,A -85,B 0,C 180,E1 19812.952,E2 19812.952} C_VEL
LIN {X 0,Y 401.499,Z 684.723,A -85,B 0,C 180,E1 19809.027,E2 19809.027} C_VEL
LIN {X 0,Y 401.499,Z 684.716,A -85,B 0,C 180,E1 19805.065,E2 19805.065} C_VEL
LIN {X 0,Y 401.5,Z 684.703,A -85,B 0,C 180,E1 19801.142,E2 19801.142} C_VEL
LIN {X 0,Y 401.499,Z 684.7,A -85,B 0,C 180,E1 19797.288,E2 19797.288} C_VEL
LIN {X 0,Y 401.496,Z 684.706,A -85,B 0,C 180,E1 19793.279,E2 19793.279} C_VEL
LIN {X 0,Y 401.491,Z 684.712,A -85,B 0,C 180,E1 19789.236,E2 19789.236} C_VEL
LIN {X 0,Y 401.497,Z 684.696,A -85,B 0,C 180,E1 19785.285,E2 19785.285} C_VEL
LIN {X 0,Y 401.491,Z 684.681,A -85,B 0,C 180,E1 19781.412,E2 19781.412} C_VEL
LIN {X 0,Y 401.491,Z 684.718,A -85,B 0,C 180,E1 19777.449,E2 19777.449} C_VEL
LIN {X 0,Y 401.496,Z 684.709,A -85,B 0,C 180,E1 19773.528,E2 19773.528} C_VEL
LIN {X 0,Y 401.498,Z 684.743,A -85,B 0,C 180,E1 19769.633,E2 19769.633} C_VEL
LIN {X 0,Y 401.586,Z 685.234,A -85,B 0,C 180,E1 19769.198,E2 19769.198} C_VEL
LIN {X 0,Y 403.09,Z 688.602,A -85,B 0,C 180,E1 19768.441,E2 19768.441} C_VEL
LIN {X 0,Y 404.18,Z 690.175,A -85,B 0,C 180,E1 19768.036,E2 19768.036} C_VEL
LIN {X 0,Y 406.155,Z 693.908,A -85,B 0,C 180,E1 19767.209,E2 19767.209} C_VEL
LIN {X 0,Y 411.97,Z 705.155,A -85,B 0,C 180,E1 19764.873,E2 19764.873} C_VEL
LIN {X 0,Y 418.066,Z 717.383,A -85,B 0,C 180,E1 19762.56,E2 19762.56} C_VEL
LIN {X 0,Y 425.492,Z 733.307,A -85,B 0,C 180,E1 19759.897,E2 19759.897} C_VEL
LIN {X 0,Y 436.409,Z 752.425,A -85,B 0,C 180,E1 19757.833,E2 19757.833} C_VEL
LIN {X 0,Y 437.725,Z 755.182,A -85,B 0,C 180,E1 19757.587,E2 19757.587} C_VEL
LIN {X 0,Y 442.76,Z 797.807,A -85,B 0,C 180,E1 19755.947,E2 19755.947} C_VEL
LIN {X 0,Y 435.515,Z 1024.723,A -85,B 0,C 180,E1 19751.873,E2 19751.873} C_VEL
LIN {X 0,Y 434.223,Z 1054.212,A -85,B 0,C 180,E1 19751.281,E2 19751.281} C_VEL
LIN {X 0,Y 432.236,Z 1076.437,A -85,B 0,C 180,E1 19750.646,E2 19750.646} C_VEL
LIN {X 0,Y 429.768,Z 1097.159,A -85,B 0,C 180,E1 19749.828,E2 19749.828} C_VEL
LIN {X 0,Y 426.795,Z 1118.853,A -85,B 0,C 180,E1 19748.718,E2 19748.718} C_VEL
LIN {X 0,Y 423.753,Z 1139.052,A -85,B 0,C 180,E1 19747.432,E2 19747.432} C_VEL
LIN {X 0,Y 420.424,Z 1158.875,A -85,B 0,C 180,E1 19745.889,E2 19745.889} C_VEL
LIN {X 0,Y 417.005,Z 1178.644,A -85,B 0,C 180,E1 19744.045,E2 19744.045} C_VEL
LIN {X 0,Y 413.771,Z 1196.964,A -85,B 0,C 180,E1 19742.032,E2 19742.032} C_VEL
LIN {X 0,Y 410.72,Z 1214.401,A -85,B 0,C 180,E1 19739.776,E2 19739.776} C_VEL
LIN {X 0,Y 408.075,Z 1229.923,A -85,B 0,C 180,E1 19737.427,E2 19737.427} C_VEL
LIN {X 0,Y 405.693,Z 1245.077,A -85,B 0,C 180,E1 19734.769,E2 19734.769} C_VEL
LIN {X 0,Y 403.75,Z 1258.758,A -85,B 0,C 180,E1 19731.958,E2 19731.958} C_VEL
LIN {X 0,Y 402.341,Z 1270.25,A -85,B 0,C 180,E1 19729.149,E2 19729.149} C_VEL
LIN {X 0,Y 401.29,Z 1280.888,A -85,B 0,C 180,E1 19726.055,E2 19726.055} C_VEL
LIN {X 0,Y 400.685,Z 1289.164,A -85,B 0,C 180,E1 19723.125,E2 19723.125} C_VEL
LIN {X 0,Y 400.384,Z 1295.565,A -85,B 0,C 180,E1 19720.212,E2 19720.212} C_VEL
LIN {X 0,Y 400.246,Z 1300.6,A -85,B 0,C 180,E1 19717.175,E2 19717.175} C_VEL
LIN {X 0,Y 400.228,Z 1303.584,A -85,B 0,C 180,E1 19714.442,E2 19714.442} C_VEL
LIN {X 0,Y 400.231,Z 1305.273,A -85,B 0,C 180,E1 19711.431,E2 19711.431} C_VEL
LIN {X 0,Y 400.236,Z 1305.326,A -85,B 0,C 180,E1 19708.855,E2 19708.855} C_VEL
LIN {X 0,Y 400.218,Z 1303.96,A -85,B 0,C 180,E1 19705.989,E2 19705.989} C_VEL
LIN {X 0,Y 400.25,Z 1301.14,A -85,B 0,C 180,E1 19703.258,E2 19703.258} C_VEL
LIN {X 0,Y 400.341,Z 1296.412,A -85,B 0,C 180,E1 19700.222,E2 19700.222} C_VEL
LIN {X 0,Y 400.619,Z 1290.541,A -85,B 0,C 180,E1 19697.46,E2 19697.46} C_VEL
LIN {X 0,Y 401.183,Z 1282.234,A -85,B 0,C 180,E1 19694.386,E2 19694.386} C_VEL
LIN {X 0,Y 402.103,Z 1272.507,A -85,B 0,C 180,E1 19691.442,E2 19691.442} C_VEL
LIN {X 0,Y 403.428,Z 1261.302,A -85,B 0,C 180,E1 19688.635,E2 19688.635} C_VEL
LIN {X 0,Y 405.243,Z 1248.119,A -85,B 0,C 180,E1 19685.823,E2 19685.823} C_VEL
LIN {X 0,Y 407.503,Z 1233.556,A -85,B 0,C 180,E1 19683.163,E2 19683.163} C_VEL
LIN {X 0,Y 410.178,Z 1217.483,A -85,B 0,C 180,E1 19680.663,E2 19680.663} C_VEL
LIN {X 0,Y 413.086,Z 1200.712,A -85,B 0,C 180,E1 19678.429,E2 19678.429} C_VEL
LIN {X 0,Y 416.286,Z 1182.847,A -85,B 0,C 180,E1 19676.385,E2 19676.385} C_VEL
LIN {X 0,Y 419.593,Z 1163.766,A -85,B 0,C 180,E1 19674.534,E2 19674.534} C_VEL
LIN {X 0,Y 422.93,Z 1143.9,A -85,B 0,C 180,E1 19672.927,E2 19672.927} C_VEL
LIN {X 0,Y 426.245,Z 1122.675,A -85,B 0,C 180,E1 19671.508,E2 19671.508} C_VEL
LIN {X 0,Y 429.189,Z 1101.724,A -85,B 0,C 180,E1 19670.378,E2 19670.378} C_VEL
LIN {X 0,Y 431.807,Z 1079.932,A -85,B 0,C 180,E1 19669.481,E2 19669.481} C_VEL
LIN {X 0,Y 434.023,Z 1056.734,A -85,B 0,C 180,E1 19668.783,E2 19668.783} C_VEL
LIN {X 0,Y 435.241,Z 1033.209,A -85,B 0,C 180,E1 19668.281,E2 19668.281} C_VEL
LIN {X 0,Y 442.28,Z 811.229,A -85,B 0,C 180,E1 19664.298,E2 19664.298} C_VEL
LIN {X 0,Y 442.627,Z 795.504,A -85,B 0,C 180,E1 19663.991,E2 19663.991} C_VEL
LIN {X 0,Y 437.491,Z 754.372,A -85,B 0,C 180,E1 19662.37,E2 19662.37} C_VEL
LIN {X 0,Y 426.2,Z 734.622,A -85,B 0,C 180,E1 19660.264,E2 19660.264} C_VEL
LIN {X 0,Y 424.55,Z 731.379,A -85,B 0,C 180,E1 19659.835,E2 19659.835} C_VEL
LIN {X 0,Y 416.862,Z 714.834,A -85,B 0,C 180,E1 19656.995,E2 19656.995} C_VEL
LIN {X 0,Y 410.516,Z 702.308,A -85,B 0,C 180,E1 19654.576,E2 19654.576} C_VEL
LIN {X 0,Y 406.109,Z 693.85,A -85,B 0,C 180,E1 19652.796,E2 19652.796} C_VEL
LIN {X 0,Y 403.423,Z 689.014,A -85,B 0,C 180,E1 19651.697,E2 19651.697} C_VEL
LIN {X 0,Y 401.799,Z 686.113,A -85,B 0,C 180,E1 19651.004,E2 19651.004} C_VEL
LIN {X 0,Y 401.534,Z 684.927,A -85,B 0,C 180,E1 19650.695,E2 19650.695} C_VEL
LIN {X 0,Y 401.494,Z 684.723,A -85,B 0,C 180,E1 19646.936,E2 19646.936} C_VEL
LIN {X 0,Y 401.499,Z 684.704,A -85,B 0,C 180,E1 19643.015,E2 19643.015} C_VEL
LIN {X 0,Y 401.491,Z 684.68,A -85,B 0,C 180,E1 19639.04,E2 19639.04} C_VEL
LIN {X 0,Y 401.492,Z 684.71,A -85,B 0,C 180,E1 19635.158,E2 19635.158} C_VEL
LIN {X 0,Y 401.494,Z 684.702,A -85,B 0,C 180,E1 19631.138,E2 19631.138} C_VEL
LIN {X 0,Y 401.51,Z 684.7,A -85,B 0,C 180,E1 19627.152,E2 19627.152} C_VEL
LIN {X 0,Y 401.495,Z 684.702,A -85,B 0,C 180,E1 19623.14,E2 19623.14} C_VEL
LIN {X 0,Y 401.496,Z 684.708,A -85,B 0,C 180,E1 19619.144,E2 19619.144} C_VEL
LIN {X 0,Y 401.497,Z 684.722,A -85,B 0,C 180,E1 19615.143,E2 19615.143} C_VEL
LIN {X 0,Y 401.492,Z 684.722,A -85,B 0,C 180,E1 19611.262,E2 19611.262} C_VEL
LIN {X 0,Y 401.495,Z 684.713,A -85,B 0,C 180,E1 19607.341,E2 19607.341} C_VEL
LIN {X 0,Y 401.505,Z 684.703,A -85,B 0,C 180,E1 19603.481,E2 19603.481} C_VEL
LIN {X 0,Y 401.505,Z 684.701,A -85,B 0,C 180,E1 19599.442,E2 19599.442} C_VEL
LIN {X 0,Y 401.502,Z 684.702,A -85,B 0,C 180,E1 19595.582,E2 19595.582} C_VEL
LIN {X 0,Y 401.495,Z 684.668,A -85,B 0,C 180,E1 19591.598,E2 19591.598} C_VEL
LIN {X 0,Y 401.487,Z 684.681,A -85,B 0,C 180,E1 19587.626,E2 19587.626} C_VEL
LIN {X 0,Y 401.491,Z 684.658,A -85,B 0,C 180,E1 19583.79,E2 19583.79} C_VEL
LIN {X 0,Y 401.51,Z 684.813,A -85,B 0,C 180,E1 19583.067,E2 19583.067} C_VEL
LIN {X 0,Y 401.837,Z 686.179,A -85,B 0,C 180,E1 19582.728,E2 19582.728} C_VEL
LIN {X 0,Y 403.646,Z 689.203,A -85,B 0,C 180,E1 19582.277,E2 19582.277} C_VEL
LIN {X 0,Y 405.893,Z 691.172,A -85,B 0,C 180,E1 19581.793,E2 19581.793} C_VEL
LIN {X 0,Y 408.352,Z 694.991,A -85,B 0,C 180,E1 19581.229,E2 19581.229} C_VEL
LIN {X 0,Y 410.43,Z 697.266,A -85,B 0,C 180,E1 19580.789,E2 19580.789} C_VEL
LIN {X 0,Y 413.742,Z 701.557,A -85,B 0,C 180,E1 19580.088,E2 19580.088} C_VEL
LIN {X 0,Y 425.332,Z 717.292,A -85,B 0,C 180,E1 19577.776,E2 19577.776} C_VEL
LIN {X 0,Y 437.409,Z 734.942,A -85,B 0,C 180,E1 19575.569,E2 19575.569} C_VEL
LIN {X 0,Y 442.899,Z 743.735,A -85,B 0,C 180,E1 19574.616,E2 19574.616} C_VEL
LIN {X 0,Y 436.503,Z 931.288,A -85,B 0,C 180,E1 19571.199,E2 19571.199} C_VEL
LIN {X 0,Y 435.234,Z 952.948,A -85,B 0,C 180,E1 19570.572,E2 19570.572} C_VEL
LIN {X 0,Y 433.428,Z 974.273,A -85,B 0,C 180,E1 19569.716,E2 19569.716} C_VEL
LIN {X 0,Y 431.332,Z 993,A -85,B 0,C 180,E1 19568.745,E2 19568.745} C_VEL
LIN {X 0,Y 428.663,Z 1012.384,A -85,B 0,C 180,E1 19567.5,E2 19567.5} C_VEL
LIN {X 0,Y 425.818,Z 1030.337,A -85,B 0,C 180,E1 19566.111,E2 19566.111} C_VEL
LIN {X 0,Y 422.55,Z 1048.193,A -85,B 0,C 180,E1 19564.438,E2 19564.438} C_VEL
LIN {X 0,Y 419.167,Z 1065.228,A -85,B 0,C 180,E1 19562.539,E2 19562.539} C_VEL
LIN {X 0,Y 415.878,Z 1080.887,A -85,B 0,C 180,E1 19560.482,E2 19560.482} C_VEL
LIN {X 0,Y 414.612,Z 1086.579,A -85,B 0,C 180,E1 19559.633,E2 19559.633} C_VEL
LIN {X 0,Y 412.645,Z 1091.902,A -85,B 0,C 180,E1 19558.897,E2 19558.897} C_VEL
LIN {X 0,Y 404.552,Z 1105.269,A -85,B 0,C 180,E1 19557.117,E2 19557.117} C_VEL
LIN {X 0,Y 402.584,Z 1109.945,A -85,B 0,C 180,E1 19556.286,E2 19556.286} C_VEL
LIN {X 0,Y 399.789,Z 1122.145,A -85,B 0,C 180,E1 19553.587,E2 19553.587} C_VEL
LIN {X 0,Y 397.448,Z 1132.708,A -85,B 0,C 180,E1 19550.775,E2 19550.775} C_VEL
LIN {X 0,Y 395.555,Z 1141.901,A -85,B 0,C 180,E1 19547.809,E2 19547.809} C_VEL
LIN {X 0,Y 394.199,Z 1149.741,A -85,B 0,C 180,E1 19544.693,E2 19544.693} C_VEL
LIN {X 0,Y 393.306,Z 1155.878,A -85,B 0,C 180,E1 19541.585,E2 19541.585} C_VEL
LIN {X 0,Y 392.798,Z 1160.368,A -85,B 0,C 180,E1 19538.49,E2 19538.49} C_VEL
LIN {X 0,Y 392.512,Z 1163.592,A -85,B 0,C 180,E1 19535.261,E2 19535.261} C_VEL
LIN {X 0,Y 392.426,Z 1165.249,A -85,B 0,C 180,E1 19532.19,E2 19532.19} C_VEL
LIN {X 0,Y 392.412,Z 1165.522,A -85,B 0,C 180,E1 19529.124,E2 19529.124} C_VEL
LIN {X 0,Y 392.468,Z 1164.559,A -85,B 0,C 180,E1 19526.056,E2 19526.056} C_VEL
LIN {X 0,Y 392.639,Z 1162.115,A -85,B 0,C 180,E1 19522.979,E2 19522.979} C_VEL
LIN {X 0,Y 393.029,Z 1158.103,A -85,B 0,C 180,E1 19519.742,E2 19519.742} C_VEL
LIN {X 0,Y 393.771,Z 1152.571,A -85,B 0,C 180,E1 19516.535,E2 19516.535} C_VEL
LIN {X 0,Y 394.938,Z 1145.35,A -85,B 0,C 180,E1 19513.377,E2 19513.377} C_VEL
LIN {X 0,Y 396.564,Z 1136.871,A -85,B 0,C 180,E1 19510.408,E2 19510.408} C_VEL
LIN {X 0,Y 398.658,Z 1127.172,A -85,B 0,C 180,E1 19507.591,E2 19507.591} C_VEL
LIN {X 0,Y 401.321,Z 1115.482,A -85,B 0,C 180,E1 19504.785,E2 19504.785} C_VEL
LIN {X 0,Y 404.204,Z 1103.078,A -85,B 0,C 180,E1 19502.288,E2 19502.288} C_VEL
LIN {X 0,Y 407.517,Z 1089.039,A -85,B 0,C 180,E1 19499.885,E2 19499.885} C_VEL
LIN {X 0,Y 410.922,Z 1074.039,A -85,B 0,C 180,E1 19497.719,E2 19497.719} C_VEL
LIN {X 0,Y 414.446,Z 1057.579,A -85,B 0,C 180,E1 19495.715,E2 19495.715} C_VEL
LIN {X 0,Y 417.886,Z 1040.371,A -85,B 0,C 180,E1 19493.944,E2 19493.944} C_VEL
LIN {X 0,Y 421.075,Z 1022.35,A -85,B 0,C 180,E1 19492.393,E2 19492.393} C_VEL
LIN {X 0,Y 423.957,Z 1003.592,A -85,B 0,C 180,E1 19491.061,E2 19491.061} C_VEL
LIN {X 0,Y 426.557,Z 983.709,A -85,B 0,C 180,E1 19489.909,E2 19489.909} C_VEL
LIN {X 0,Y 428.543,Z 963.988,A -85,B 0,C 180,E1 19489.013,E2 19489.013} C_VEL
LIN {X 0,Y 430.111,Z 942.286,A -85,B 0,C 180,E1 19488.271,E2 19488.271} C_VEL
LIN {X 0,Y 431.051,Z 920.717,A -85,B 0,C 180,E1 19487.758,E2 19487.758} C_VEL
LIN {X 0,Y 437.147,Z 746.984,A -85,B 0,C 180,E1 19484.58,E2 19484.58} C_VEL
LIN {X 0,Y 426.238,Z 730.38,A -85,B 0,C 180,E1 19482.591,E2 19482.591} C_VEL
LIN {X 0,Y 416.336,Z 716.419,A -85,B 0,C 180,E1 19480.649,E2 19480.649} C_VEL
LIN {X 0,Y 409.39,Z 707.165,A -85,B 0,C 180,E1 19479.194,E2 19479.194} C_VEL
LIN {X 0,Y 405.734,Z 702.358,A -85,B 0,C 180,E1 19478.39,E2 19478.39} C_VEL
LIN {X 0,Y 402.559,Z 698.012,A -85,B 0,C 180,E1 19477.662,E2 19477.662} C_VEL
LIN {X 0,Y 398.924,Z 693.827,A -85,B 0,C 180,E1 19476.823,E2 19476.823} C_VEL
LIN {X 0,Y 397.613,Z 691.677,A -85,B 0,C 180,E1 19476.493,E2 19476.493} C_VEL
LIN {X 0,Y 394.857,Z 689.136,A -85,B 0,C 180,E1 19475.844,E2 19475.844} C_VEL
LIN {X 0,Y 393.698,Z 686.491,A -85,B 0,C 180,E1 19475.442,E2 19475.442} C_VEL
LIN {X 0,Y 393.562,Z 685.719,A -85,B 0,C 180,E1 19475.041,E2 19475.041} C_VEL
LIN {X 0,Y 393.553,Z 685.637,A -85,B 0,C 180,E1 19471.047,E2 19471.047} C_VEL
LIN {X 0,Y 393.559,Z 685.698,A -85,B 0,C 180,E1 19467.05,E2 19467.05} C_VEL
LIN {X 0,Y 393.566,Z 685.703,A -85,B 0,C 180,E1 19463.032,E2 19463.032} C_VEL
LIN {X 0,Y 393.56,Z 685.702,A -85,B 0,C 180,E1 19458.977,E2 19458.977} C_VEL
LIN {X 0,Y 393.553,Z 685.696,A -85,B 0,C 180,E1 19455.019,E2 19455.019} C_VEL
LIN {X 0,Y 393.553,Z 685.69,A -85,B 0,C 180,E1 19450.985,E2 19450.985} C_VEL
LIN {X 0,Y 393.564,Z 685.686,A -85,B 0,C 180,E1 19447.005,E2 19447.005} C_VEL
LIN {X 0,Y 393.559,Z 685.693,A -85,B 0,C 180,E1 19442.913,E2 19442.913} C_VEL
LIN {X 0,Y 393.56,Z 685.705,A -85,B 0,C 180,E1 19438.836,E2 19438.836} C_VEL
LIN {X 0,Y 393.561,Z 685.713,A -85,B 0,C 180,E1 19434.753,E2 19434.753} C_VEL
LIN {X 0,Y 393.563,Z 685.707,A -85,B 0,C 180,E1 19430.79,E2 19430.79} C_VEL
LIN {X 0,Y 393.553,Z 685.663,A -85,B 0,C 180,E1 19426.782,E2 19426.782} C_VEL
LIN {X 0,Y 393.552,Z 685.694,A -85,B 0,C 180,E1 19422.792,E2 19422.792} C_VEL
LIN {X 0,Y 393.556,Z 685.701,A -85,B 0,C 180,E1 19418.697,E2 19418.697} C_VEL
LIN {X 0,Y 393.555,Z 685.674,A -85,B 0,C 180,E1 19414.735,E2 19414.735} C_VEL
LIN {X 0,Y 393.588,Z 685.936,A -85,B 0,C 180,E1 19410.788,E2 19410.788} C_VEL
LIN {X 0,Y 395.04,Z 689.424,A -85,B 0,C 180,E1 19409.925,E2 19409.925} C_VEL
LIN {X 0,Y 396.411,Z 691.492,A -85,B 0,C 180,E1 19409.37,E2 19409.37} C_VEL
LIN {X 0,Y 398.335,Z 695.032,A -85,B 0,C 180,E1 19408.527,E2 19408.527} C_VEL
LIN {X 0,Y 403.977,Z 705.685,A -85,B 0,C 180,E1 19406.16,E2 19406.16} C_VEL
LIN {X 0,Y 410.552,Z 718.841,A -85,B 0,C 180,E1 19403.542,E2 19403.542} C_VEL
LIN {X 0,Y 416.355,Z 730.969,A -85,B 0,C 180,E1 19401.408,E2 19401.408} C_VEL
LIN {X 0,Y 426.703,Z 748.381,A -85,B 0,C 180,E1 19399.33,E2 19399.33} C_VEL
LIN {X 0,Y 432.462,Z 759.11,A -85,B 0,C 180,E1 19398.23,E2 19398.23} C_VEL
LIN {X 0,Y 437.049,Z 799.13,A -85,B 0,C 180,E1 19396.663,E2 19396.663} C_VEL
LIN {X 0,Y 429.432,Z 1025.759,A -85,B 0,C 180,E1 19392.551,E2 19392.551} C_VEL
LIN {X 0,Y 428.113,Z 1053.451,A -85,B 0,C 180,E1 19391.981,E2 19391.981} C_VEL
LIN {X 0,Y 426.022,Z 1075.646,A -85,B 0,C 180,E1 19391.335,E2 19391.335} C_VEL
LIN {X 0,Y 423.438,Z 1096.381,A -85,B 0,C 180,E1 19390.507,E2 19390.507} C_VEL
LIN {X 0,Y 420.292,Z 1118.05,A -85,B 0,C 180,E1 19389.383,E2 19389.383} C_VEL
LIN {X 0,Y 416.981,Z 1138.724,A -85,B 0,C 180,E1 19388.041,E2 19388.041} C_VEL
LIN {X 0,Y 413.545,Z 1158.25,A -85,B 0,C 180,E1 19386.495,E2 19386.495} C_VEL
LIN {X 0,Y 410.079,Z 1177.094,A -85,B 0,C 180,E1 19384.71,E2 19384.71} C_VEL
LIN {X 0,Y 406.674,Z 1195.384,A -85,B 0,C 180,E1 19382.673,E2 19382.673} C_VEL
LIN {X 0,Y 403.396,Z 1212.91,A -85,B 0,C 180,E1 19380.372,E2 19380.372} C_VEL
LIN {X 0,Y 400.513,Z 1228.918,A -85,B 0,C 180,E1 19377.904,E2 19377.904} C_VEL
LIN {X 0,Y 397.935,Z 1244.35,A -85,B 0,C 180,E1 19375.127,E2 19375.127} C_VEL
LIN {X 0,Y 395.902,Z 1257.935,A -85,B 0,C 180,E1 19372.26,E2 19372.26} C_VEL
LIN {X 0,Y 394.435,Z 1269.349,A -85,B 0,C 180,E1 19369.394,E2 19369.394} C_VEL
LIN {X 0,Y 393.398,Z 1279.437,A -85,B 0,C 180,E1 19366.386,E2 19366.386} C_VEL
LIN {X 0,Y 392.762,Z 1287.727,A -85,B 0,C 180,E1 19363.394,E2 19363.394} C_VEL
LIN {X 0,Y 392.462,Z 1294.144,A -85,B 0,C 180,E1 19360.421,E2 19360.421} C_VEL
LIN {X 0,Y 392.334,Z 1299.193,A -85,B 0,C 180,E1 19357.321,E2 19357.321} C_VEL
LIN {X 0,Y 392.336,Z 1302.187,A -85,B 0,C 180,E1 19354.531,E2 19354.531} C_VEL
LIN {X 0,Y 392.348,Z 1303.854,A -85,B 0,C 180,E1 19351.606,E2 19351.606} C_VEL
LIN {X 0,Y 392.357,Z 1303.962,A -85,B 0,C 180,E1 19348.978,E2 19348.978} C_VEL
LIN {X 0,Y 392.327,Z 1302.69,A -85,B 0,C 180,E1 19346.054,E2 19346.054} C_VEL
LIN {X 0,Y 392.345,Z 1299.736,A -85,B 0,C 180,E1 19343.121,E2 19343.121} C_VEL
LIN {X 0,Y 392.425,Z 1294.995,A -85,B 0,C 180,E1 19340.023,E2 19340.023} C_VEL
LIN {X 0,Y 392.689,Z 1289.107,A -85,B 0,C 180,E1 19337.202,E2 19337.202} C_VEL
LIN {X 0,Y 393.272,Z 1280.783,A -85,B 0,C 180,E1 19334.064,E2 19334.064} C_VEL
LIN {X 0,Y 394.243,Z 1271.042,A -85,B 0,C 180,E1 19331.058,E2 19331.058} C_VEL
LIN {X 0,Y 395.641,Z 1259.824,A -85,B 0,C 180,E1 19328.193,E2 19328.193} C_VEL
LIN {X 0,Y 397.579,Z 1246.633,A -85,B 0,C 180,E1 19325.326,E2 19325.326} C_VEL
LIN {X 0,Y 399.987,Z 1232.065,A -85,B 0,C 180,E1 19322.617,E2 19322.617} C_VEL
LIN {X 0,Y 402.84,Z 1215.991,A -85,B 0,C 180,E1 19320.075,E2 19320.075} C_VEL
LIN {X 0,Y 405.963,Z 1198.995,A -85,B 0,C 180,E1 19317.778,E2 19317.778} C_VEL
LIN {X 0,Y 409.43,Z 1180.658,A -85,B 0,C 180,E1 19315.66,E2 19315.66} C_VEL
LIN {X 0,Y 412.952,Z 1161.519,A -85,B 0,C 180,E1 19313.789,E2 19313.789} C_VEL
LIN {X 0,Y 416.332,Z 1142.43,A -85,B 0,C 180,E1 19312.238,E2 19312.238} C_VEL
LIN {X 0,Y 419.689,Z 1122.009,A -85,B 0,C 180,E1 19310.853,E2 19310.853} C_VEL
LIN {X 0,Y 422.808,Z 1100.917,A -85,B 0,C 180,E1 19309.702,E2 19309.702} C_VEL
LIN {X 0,Y 425.537,Z 1079.479,A -85,B 0,C 180,E1 19308.806,E2 19308.806} C_VEL
LIN {X 0,Y 427.894,Z 1056.112,A -85,B 0,C 180,E1 19308.089,E2 19308.089} C_VEL
LIN {X 0,Y 429.174,Z 1033.194,A -85,B 0,C 180,E1 19307.586,E2 19307.586} C_VEL
LIN {X 0,Y 436.611,Z 810.639,A -85,B 0,C 180,E1 19303.55,E2 19303.55} C_VEL
LIN {X 0,Y 436.91,Z 796.936,A -85,B 0,C 180,E1 19303.276,E2 19303.276} C_VEL
LIN {X 0,Y 432.232,Z 758.435,A -85,B 0,C 180,E1 19301.731,E2 19301.731} C_VEL
LIN {X 0,Y 421.188,Z 738.879,A -85,B 0,C 180,E1 19299.597,E2 19299.597} C_VEL
LIN {X 0,Y 415.541,Z 729.4,A -85,B 0,C 180,E1 19298.373,E2 19298.373} C_VEL
LIN {X 0,Y 408.759,Z 715.195,A -85,B 0,C 180,E1 19295.775,E2 19295.775} C_VEL
LIN {X 0,Y 402.911,Z 703.682,A -85,B 0,C 180,E1 19293.429,E2 19293.429} C_VEL
LIN {X 0,Y 398.281,Z 694.969,A -85,B 0,C 180,E1 19291.478,E2 19291.478} C_VEL
LIN {X 0,Y 395.721,Z 690.269,A -85,B 0,C 180,E1 19290.353,E2 19290.353} C_VEL
LIN {X 0,Y 393.833,Z 686.973,A -85,B 0,C 180,E1 19289.506,E2 19289.506} C_VEL
LIN {X 0,Y 393.579,Z 685.873,A -85,B 0,C 180,E1 19289.193,E2 19289.193} C_VEL
LIN {X 0,Y 393.555,Z 685.674,A -85,B 0,C 180,E1 19285.255,E2 19285.255} C_VEL
LIN {X 0,Y 393.556,Z 685.701,A -85,B 0,C 180,E1 19281.303,E2 19281.303} C_VEL
LIN {X 0,Y 393.552,Z 685.695,A -85,B 0,C 180,E1 19277.208,E2 19277.208} C_VEL
LIN {X 0,Y 393.553,Z 685.663,A -85,B 0,C 180,E1 19273.218,E2 19273.218} C_VEL
LIN {X 0,Y 393.563,Z 685.707,A -85,B 0,C 180,E1 19269.21,E2 19269.21} C_VEL
LIN {X 0,Y 393.56,Z 685.714,A -85,B 0,C 180,E1 19265.213,E2 19265.213} C_VEL
LIN {X 0,Y 393.557,Z 685.705,A -85,B 0,C 180,E1 19261.164,E2 19261.164} C_VEL
LIN {X 0,Y 393.559,Z 685.692,A -85,B 0,C 180,E1 19257.087,E2 19257.087} C_VEL
LIN {X 0,Y 393.564,Z 685.686,A -85,B 0,C 180,E1 19252.995,E2 19252.995} C_VEL
LIN {X 0,Y 393.553,Z 685.691,A -85,B 0,C 180,E1 19249.015,E2 19249.015} C_VEL
LIN {X 0,Y 393.553,Z 685.697,A -85,B 0,C 180,E1 19244.981,E2 19244.981} C_VEL
LIN {X 0,Y 393.558,Z 685.701,A -85,B 0,C 180,E1 19240.919,E2 19240.919} C_VEL
LIN {X 0,Y 393.566,Z 685.702,A -85,B 0,C 180,E1 19236.873,E2 19236.873} C_VEL
LIN {X 0,Y 393.564,Z 685.693,A -85,B 0,C 180,E1 19232.767,E2 19232.767} C_VEL
LIN {X 0,Y 393.554,Z 685.638,A -85,B 0,C 180,E1 19228.783,E2 19228.783} C_VEL
LIN {X 0,Y 393.576,Z 685.828,A -85,B 0,C 180,E1 19224.684,E2 19224.684} C_VEL
LIN {X 0,Y 393.935,Z 687.295,A -85,B 0,C 180,E1 19224.304,E2 19224.304} C_VEL
LIN {X 0,Y 395.808,Z 690.288,A -85,B 0,C 180,E1 19223.809,E2 19223.809} C_VEL
LIN {X 0,Y 398.134,Z 692.272,A -85,B 0,C 180,E1 19223.272,E2 19223.272} C_VEL
LIN {X 0,Y 400.609,Z 696.09,A -85,B 0,C 180,E1 19222.664,E2 19222.664} C_VEL
LIN {X 0,Y 402.691,Z 698.274,A -85,B 0,C 180,E1 19222.195,E2 19222.195} C_VEL
LIN {X 0,Y 405.955,Z 702.577,A -85,B 0,C 180,E1 19221.454,E2 19221.454} C_VEL
LIN {X 0,Y 415.103,Z 714.701,A -85,B 0,C 180,E1 19219.5,E2 19219.5} C_VEL
LIN {X 0,Y 425.767,Z 729.734,A -85,B 0,C 180,E1 19217.397,E2 19217.397} C_VEL
LIN {X 0,Y 436.297,Z 745.68,A -85,B 0,C 180,E1 19215.472,E2 19215.472} C_VEL
LIN {X 0,Y 437.213,Z 747.451,A -85,B 0,C 180,E1 19215.303,E2 19215.303} C_VEL
LIN {X 0,Y 430.585,Z 932.603,A -85,B 0,C 180,E1 19211.895,E2 19211.895} C_VEL
LIN {X 0,Y 429.271,Z 954.355,A -85,B 0,C 180,E1 19211.257,E2 19211.257} C_VEL
LIN {X 0,Y 427.397,Z 975.674,A -85,B 0,C 180,E1 19210.391,E2 19210.391} C_VEL
LIN {X 0,Y 425.137,Z 995.084,A -85,B 0,C 180,E1 19209.37,E2 19209.37} C_VEL
LIN {X 0,Y 422.44,Z 1013.782,A -85,B 0,C 180,E1 19208.151,E2 19208.151} C_VEL
LIN {X 0,Y 419.473,Z 1031.734,A -85,B 0,C 180,E1 19206.746,E2 19206.746} C_VEL
LIN {X 0,Y 416.061,Z 1049.592,A -85,B 0,C 180,E1 19205.053,E2 19205.053} C_VEL
LIN {X 0,Y 412.52,Z 1066.629,A -85,B 0,C 180,E1 19203.13,E2 19203.13} C_VEL
LIN {X 0,Y 409.07,Z 1082.289,A -85,B 0,C 180,E1 19201.045,E2 19201.045} C_VEL
LIN {X 0,Y 405.665,Z 1096.916,A -85,B 0,C 180,E1 19198.725,E2 19198.725} C_VEL
LIN {X 0,Y 402.584,Z 1109.945,A -85,B 0,C 180,E1 19196.286,E2 19196.286} C_VEL
LIN {X 0,Y 400.658,Z 1114.577,A -85,B 0,C 180,E1 19195.431,E2 19195.431} C_VEL
LIN {X 0,Y 392.793,Z 1126.063,A -85,B 0,C 180,E1 19193.338,E2 19193.338} C_VEL
LIN {X 0,Y 390.976,Z 1129.934,A -85,B 0,C 180,E1 19192.392,E2 19192.392} C_VEL
LIN {X 0,Y 388.733,Z 1139.873,A -85,B 0,C 180,E1 19189.377,E2 19189.377} C_VEL
LIN {X 0,Y 387.066,Z 1147.994,A -85,B 0,C 180,E1 19186.353,E2 19186.353} C_VEL
LIN {X 0,Y 385.887,Z 1154.843,A -85,B 0,C 180,E1 19183.18,E2 19183.18} C_VEL
LIN {X 0,Y 385.174,Z 1160.04,A -85,B 0,C 180,E1 19180.016,E2 19180.016} C_VEL
LIN {X 0,Y 384.773,Z 1163.699,A -85,B 0,C 180,E1 19176.865,E2 19176.865} C_VEL
LIN {X 0,Y 384.584,Z 1166.045,A -85,B 0,C 180,E1 19173.727,E2 19173.727} C_VEL
LIN {X 0,Y 384.529,Z 1166.941,A -85,B 0,C 180,E1 19170.596,E2 19170.596} C_VEL
LIN {X 0,Y 384.555,Z 1166.496,A -85,B 0,C 180,E1 19167.318,E2 19167.318} C_VEL
LIN {X 0,Y 384.695,Z 1164.751,A -85,B 0,C 180,E1 19164.182,E2 19164.182} C_VEL
LIN {X 0,Y 385.003,Z 1161.514,A -85,B 0,C 180,E1 19161.036,E2 19161.036} C_VEL
LIN {X 0,Y 385.613,Z 1156.63,A -85,B 0,C 180,E1 19157.725,E2 19157.725} C_VEL
LIN {X 0,Y 386.668,Z 1150.387,A -85,B 0,C 180,E1 19154.554,E2 19154.554} C_VEL
LIN {X 0,Y 388.198,Z 1142.309,A -85,B 0,C 180,E1 19151.375,E2 19151.375} C_VEL
LIN {X 0,Y 390.282,Z 1132.851,A -85,B 0,C 180,E1 19148.352,E2 19148.352} C_VEL
LIN {X 0,Y 392.876,Z 1122.072,A -85,B 0,C 180,E1 19145.492,E2 19145.492} C_VEL
LIN {X 0,Y 395.873,Z 1109.839,A -85,B 0,C 180,E1 19142.797,E2 19142.797} C_VEL
LIN {X 0,Y 399.229,Z 1096.212,A -85,B 0,C 180,E1 19140.273,E2 19140.273} C_VEL
LIN {X 0,Y 402.9,Z 1081.203,A -85,B 0,C 180,E1 19137.923,E2 19137.923} C_VEL
LIN {X 0,Y 406.451,Z 1065.788,A -85,B 0,C 180,E1 19135.885,E2 19135.885} C_VEL
LIN {X 0,Y 410.05,Z 1048.956,A -85,B 0,C 180,E1 19134.011,E2 19134.011} C_VEL
LIN {X 0,Y 413.635,Z 1030.657,A -85,B 0,C 180,E1 19132.299,E2 19132.299} C_VEL
LIN {X 0,Y 416.762,Z 1012.352,A -85,B 0,C 180,E1 19130.88,E2 19130.88} C_VEL
LIN {X 0,Y 419.479,Z 993.401,A -85,B 0,C 180,E1 19129.675,E2 19129.675} C_VEL
LIN {X 0,Y 421.882,Z 972.999,A -85,B 0,C 180,E1 19128.631,E2 19128.631} C_VEL
LIN {X 0,Y 423.708,Z 951.954,A -85,B 0,C 180,E1 19127.815,E2 19127.815} C_VEL
LIN {X 0,Y 424.897,Z 930.567,A -85,B 0,C 180,E1 19127.223,E2 19127.223} C_VEL
LIN {X 0,Y 431.535,Z 750.587,A -85,B 0,C 180,E1 19123.871,E2 19123.871} C_VEL
LIN {X 0,Y 420.231,Z 733.372,A -85,B 0,C 180,E1 19121.729,E2 19121.729} C_VEL
LIN {X 0,Y 409.692,Z 718.639,A -85,B 0,C 180,E1 19119.567,E2 19119.567} C_VEL
LIN {X 0,Y 402.12,Z 708.675,A -85,B 0,C 180,E1 19117.891,E2 19117.891} C_VEL
LIN {X 0,Y 398.185,Z 703.579,A -85,B 0,C 180,E1 19116.97,E2 19116.97} C_VEL
LIN {X 0,Y 394.991,Z 699.282,A -85,B 0,C 180,E1 19116.188,E2 19116.188} C_VEL
LIN {X 0,Y 391.294,Z 695.16,A -85,B 0,C 180,E1 19115.274,E2 19115.274} C_VEL
LIN {X 0,Y 389.861,Z 692.784,A -85,B 0,C 180,E1 19114.884,E2 19114.884} C_VEL
LIN {X 0,Y 387.081,Z 690.393,A -85,B 0,C 180,E1 19114.182,E2 19114.182} C_VEL
LIN {X 0,Y 385.749,Z 687.445,A -85,B 0,C 180,E1 19113.689,E2 19113.689} C_VEL
LIN {X 0,Y 385.626,Z 686.755,A -85,B 0,C 180,E1 19113.345,E2 19113.345} C_VEL
LIN {X 0,Y 385.616,Z 686.62,A -85,B 0,C 180,E1 19109.344,E2 19109.344} C_VEL
LIN {X 0,Y 385.621,Z 686.685,A -85,B 0,C 180,E1 19105.33,E2 19105.33} C_VEL
LIN {X 0,Y 385.619,Z 686.685,A -85,B 0,C 180,E1 19101.285,E2 19101.285} C_VEL
LIN {X 0,Y 385.616,Z 686.689,A -85,B 0,C 180,E1 19097.193,E2 19097.193} C_VEL
LIN {X 0,Y 385.618,Z 686.699,A -85,B 0,C 180,E1 19093.19,E2 19093.19} C_VEL
LIN {X 0,Y 385.623,Z 686.701,A -85,B 0,C 180,E1 19089.101,E2 19089.101} C_VEL
LIN {X 0,Y 385.621,Z 686.693,A -85,B 0,C 180,E1 19085.058,E2 19085.058} C_VEL
LIN {X 0,Y 385.62,Z 686.681,A -85,B 0,C 180,E1 19081.04,E2 19081.04} C_VEL
LIN {X 0,Y 385.62,Z 686.676,A -85,B 0,C 180,E1 19077.028,E2 19077.028} C_VEL
LIN {X 0,Y 385.627,Z 686.678,A -85,B 0,C 180,E1 19073.001,E2 19073.001} C_VEL
LIN {X 0,Y 385.616,Z 686.679,A -85,B 0,C 180,E1 19068.938,E2 19068.938} C_VEL
LIN {X 0,Y 385.615,Z 686.683,A -85,B 0,C 180,E1 19064.819,E2 19064.819} C_VEL
LIN {X 0,Y 385.61,Z 686.654,A -85,B 0,C 180,E1 19060.774,E2 19060.774} C_VEL
LIN {X 0,Y 385.622,Z 686.673,A -85,B 0,C 180,E1 19056.79,E2 19056.79} C_VEL
LIN {X 0,Y 385.63,Z 686.76,A -85,B 0,C 180,E1 19052.683,E2 19052.683} C_VEL
LIN {X 0,Y 385.726,Z 687.333,A -85,B 0,C 180,E1 19052.271,E2 19052.271} C_VEL
LIN {X 0,Y 387.5,Z 690.903,A -85,B 0,C 180,E1 19051.319,E2 19051.319} C_VEL
LIN {X 0,Y 388.498,Z 692.363,A -85,B 0,C 180,E1 19050.895,E2 19050.895} C_VEL
LIN {X 0,Y 390.687,Z 696.333,A -85,B 0,C 180,E1 19049.882,E2 19049.882} C_VEL
LIN {X 0,Y 396.427,Z 707.167,A -85,B 0,C 180,E1 19047.334,E2 19047.334} C_VEL
LIN {X 0,Y 402.836,Z 719.82,A -85,B 0,C 180,E1 19044.668,E2 19044.668} C_VEL
LIN {X 0,Y 407.016,Z 728.328,A -85,B 0,C 180,E1 19043.085,E2 19043.085} C_VEL
LIN {X 0,Y 417.938,Z 746.17,A -85,B 0,C 180,E1 19040.745,E2 19040.745} C_VEL
LIN {X 0,Y 427.247,Z 762.885,A -85,B 0,C 180,E1 19038.893,E2 19038.893} C_VEL
LIN {X 0,Y 431.398,Z 800.719,A -85,B 0,C 180,E1 19037.393,E2 19037.393} C_VEL
LIN {X 0,Y 423.418,Z 1026.538,A -85,B 0,C 180,E1 19033.253,E2 19033.253} C_VEL
LIN {X 0,Y 422.08,Z 1052.526,A -85,B 0,C 180,E1 19032.705,E2 19032.705} C_VEL
LIN {X 0,Y 419.862,Z 1074.93,A -85,B 0,C 180,E1 19032.042,E2 19032.042} C_VEL
LIN {X 0,Y 417.221,Z 1095.209,A -85,B 0,C 180,E1 19031.224,E2 19031.224} C_VEL
LIN {X 0,Y 414.067,Z 1115.957,A -85,B 0,C 180,E1 19030.144,E2 19030.144} C_VEL
LIN {X 0,Y 410.594,Z 1136.566,A -85,B 0,C 180,E1 19028.809,E2 19028.809} C_VEL
LIN {X 0,Y 407.005,Z 1156.051,A -85,B 0,C 180,E1 19027.256,E2 19027.256} C_VEL
LIN {X 0,Y 403.191,Z 1175.685,A -85,B 0,C 180,E1 19025.382,E2 19025.382} C_VEL
LIN {X 0,Y 399.561,Z 1194.094,A -85,B 0,C 180,E1 19023.302,E2 19023.302} C_VEL
LIN {X 0,Y 396.127,Z 1211.42,A -85,B 0,C 180,E1 19020.991,E2 19020.991} C_VEL
LIN {X 0,Y 393.162,Z 1226.946,A -85,B 0,C 180,E1 19018.561,E2 19018.561} C_VEL
LIN {X 0,Y 390.45,Z 1242.104,A -85,B 0,C 180,E1 19015.806,E2 19015.806} C_VEL
LIN {X 0,Y 388.259,Z 1255.802,A -85,B 0,C 180,E1 19012.883,E2 19012.883} C_VEL
LIN {X 0,Y 386.676,Z 1267.317,A -85,B 0,C 180,E1 19009.957,E2 19009.957} C_VEL
LIN {X 0,Y 385.51,Z 1277.985,A -85,B 0,C 180,E1 19006.731,E2 19006.731} C_VEL
LIN {X 0,Y 384.845,Z 1286.304,A -85,B 0,C 180,E1 19003.669,E2 19003.669} C_VEL
LIN {X 0,Y 384.532,Z 1292.753,A -85,B 0,C 180,E1 19000.621,E2 19000.621} C_VEL
LIN {X 0,Y 384.425,Z 1297.785,A -85,B 0,C 180,E1 18997.472,E2 18997.472} C_VEL
LIN {X 0,Y 384.443,Z 1300.79,A -85,B 0,C 180,E1 18994.624,E2 18994.624} C_VEL
LIN {X 0,Y 384.468,Z 1302.463,A -85,B 0,C 180,E1 18991.639,E2 18991.639} C_VEL
LIN {X 0,Y 384.479,Z 1302.571,A -85,B 0,C 180,E1 18988.957,E2 18988.957} C_VEL
LIN {X 0,Y 384.437,Z 1301.294,A -85,B 0,C 180,E1 18985.973,E2 18985.973} C_VEL
LIN {X 0,Y 384.433,Z 1298.329,A -85,B 0,C 180,E1 18982.979,E2 18982.979} C_VEL
LIN {X 0,Y 384.509,Z 1293.576,A -85,B 0,C 180,E1 18979.816,E2 18979.816} C_VEL
LIN {X 0,Y 384.758,Z 1287.671,A -85,B 0,C 180,E1 18976.934,E2 18976.934} C_VEL
LIN {X 0,Y 385.375,Z 1279.333,A -85,B 0,C 180,E1 18973.728,E2 18973.728} C_VEL
LIN {X 0,Y 386.399,Z 1269.577,A -85,B 0,C 180,E1 18970.658,E2 18970.658} C_VEL
LIN {X 0,Y 387.876,Z 1258.338,A -85,B 0,C 180,E1 18967.731,E2 18967.731} C_VEL
LIN {X 0,Y 389.939,Z 1245.145,A -85,B 0,C 180,E1 18964.809,E2 18964.809} C_VEL
LIN {X 0,Y 392.5,Z 1230.572,A -85,B 0,C 180,E1 18962.05,E2 18962.05} C_VEL
LIN {X 0,Y 395.531,Z 1214.497,A -85,B 0,C 180,E1 18959.463,E2 18959.463} C_VEL
LIN {X 0,Y 398.908,Z 1197.289,A -85,B 0,C 180,E1 18957.105,E2 18957.105} C_VEL
LIN {X 0,Y 402.643,Z 1178.469,A -85,B 0,C 180,E1 18954.911,E2 18954.911} C_VEL
LIN {X 0,Y 406.402,Z 1159.269,A -85,B 0,C 180,E1 18953.021,E2 18953.021} C_VEL
LIN {X 0,Y 410.124,Z 1139.093,A -85,B 0,C 180,E1 18951.384,E2 18951.384} C_VEL
LIN {X 0,Y 413.679,Z 1118.221,A -85,B 0,C 180,E1 18949.992,E2 18949.992} C_VEL
LIN {X 0,Y 416.92,Z 1097.334,A -85,B 0,C 180,E1 18948.872,E2 18948.872} C_VEL
LIN {X 0,Y 419.641,Z 1076.556,A -85,B 0,C 180,E1 18948.02,E2 18948.02} C_VEL
LIN {X 0,Y 421.984,Z 1053.516,A -85,B 0,C 180,E1 18947.324,E2 18947.324} C_VEL
LIN {X 0,Y 423.296,Z 1029.471,A -85,B 0,C 180,E1 18946.804,E2 18946.804} C_VEL
LIN {X 0,Y 431.175,Z 805.81,A -85,B 0,C 180,E1 18942.705,E2 18942.705} C_VEL
LIN {X 0,Y 431.261,Z 798.321,A -85,B 0,C 180,E1 18942.54,E2 18942.54} C_VEL
LIN {X 0,Y 427.06,Z 762.532,A -85,B 0,C 180,E1 18941.081,E2 18941.081} C_VEL
LIN {X 0,Y 416.713,Z 744.055,A -85,B 0,C 180,E1 18939.016,E2 18939.016} C_VEL
LIN {X 0,Y 406.312,Z 726.998,A -85,B 0,C 180,E1 18936.725,E2 18936.725} C_VEL
LIN {X 0,Y 399.378,Z 712.947,A -85,B 0,C 180,E1 18933.937,E2 18933.937} C_VEL
LIN {X 0,Y 395.035,Z 704.651,A -85,B 0,C 180,E1 18932.108,E2 18932.108} C_VEL
LIN {X 0,Y 392.769,Z 700.41,A -85,B 0,C 180,E1 18931.116,E2 18931.116} C_VEL
LIN {X 0,Y 390.231,Z 695.767,A -85,B 0,C 180,E1 18929.975,E2 18929.975} C_VEL
LIN {X 0,Y 387.798,Z 691.259,A -85,B 0,C 180,E1 18928.825,E2 18928.825} C_VEL
LIN {X 0,Y 385.914,Z 688.068,A -85,B 0,C 180,E1 18927.937,E2 18927.937} C_VEL
LIN {X 0,Y 385.637,Z 686.801,A -85,B 0,C 180,E1 18927.54,E2 18927.54} C_VEL
LIN {X 0,Y 385.615,Z 686.668,A -85,B 0,C 180,E1 18923.534,E2 18923.534} C_VEL
LIN {X 0,Y 385.612,Z 686.656,A -85,B 0,C 180,E1 18919.541,E2 18919.541} C_VEL
LIN {X 0,Y 385.622,Z 686.693,A -85,B 0,C 180,E1 18915.489,E2 18915.489} C_VEL
LIN {X 0,Y 385.617,Z 686.668,A -85,B 0,C 180,E1 18911.456,E2 18911.456} C_VEL
LIN {X 0,Y 385.615,Z 686.677,A -85,B 0,C 180,E1 18907.449,E2 18907.449} C_VEL
LIN {X 0,Y 385.616,Z 686.68,A -85,B 0,C 180,E1 18903.409,E2 18903.409} C_VEL
LIN {X 0,Y 385.624,Z 686.688,A -85,B 0,C 180,E1 18899.405,E2 18899.405} C_VEL
LIN {X 0,Y 385.617,Z 686.701,A -85,B 0,C 180,E1 18895.389,E2 18895.389} C_VEL
LIN {X 0,Y 385.615,Z 686.7,A -85,B 0,C 180,E1 18891.35,E2 18891.35} C_VEL
LIN {X 0,Y 385.617,Z 686.69,A -85,B 0,C 180,E1 18887.268,E2 18887.268} C_VEL
LIN {X 0,Y 385.624,Z 686.681,A -85,B 0,C 180,E1 18883.273,E2 18883.273} C_VEL
LIN {X 0,Y 385.627,Z 686.678,A -85,B 0,C 180,E1 18879.193,E2 18879.193} C_VEL
LIN {X 0,Y 385.624,Z 686.679,A -85,B 0,C 180,E1 18875.157,E2 18875.157} C_VEL
LIN {X 0,Y 385.624,Z 686.628,A -85,B 0,C 180,E1 18871.166,E2 18871.166} C_VEL
LIN {X 0,Y 385.62,Z 686.667,A -85,B 0,C 180,E1 18867.146,E2 18867.146} C_VEL
LIN {X 0,Y 385.676,Z 687.066,A -85,B 0,C 180,E1 18866.303,E2 18866.303} C_VEL
LIN {X 0,Y 386.233,Z 688.914,A -85,B 0,C 180,E1 18865.944,E2 18865.944} C_VEL
LIN {X 0,Y 388.235,Z 691.657,A -85,B 0,C 180,E1 18865.398,E2 18865.398} C_VEL
LIN {X 0,Y 390.348,Z 693.343,A -85,B 0,C 180,E1 18864.874,E2 18864.874} C_VEL
LIN {X 0,Y 392.844,Z 697.178,A -85,B 0,C 180,E1 18864.214,E2 18864.214} C_VEL
LIN {X 0,Y 395.049,Z 699.4,A -85,B 0,C 180,E1 18863.683,E2 18863.683} C_VEL
LIN {X 0,Y 398.255,Z 703.649,A -85,B 0,C 180,E1 18862.902,E2 18862.902} C_VEL
LIN {X 0,Y 400.338,Z 706.448,A -85,B 0,C 180,E1 18862.409,E2 18862.409} C_VEL
LIN {X 0,Y 404.2,Z 711.388,A -85,B 0,C 180,E1 18861.528,E2 18861.528} C_VEL
LIN {X 0,Y 411.779,Z 721.519,A -85,B 0,C 180,E1 18859.884,E2 18859.884} C_VEL
LIN {X 0,Y 422.059,Z 736.163,A -85,B 0,C 180,E1 18857.808,E2 18857.808} C_VEL
LIN {X 0,Y 431.603,Z 750.885,A -85,B 0,C 180,E1 18856.013,E2 18856.013} C_VEL
LIN {X 0,Y 424.738,Z 933.813,A -85,B 0,C 180,E1 18852.612,E2 18852.612} C_VEL
LIN {X 0,Y 423.382,Z 955.635,A -85,B 0,C 180,E1 18851.965,E2 18851.965} C_VEL
LIN {X 0,Y 421.51,Z 976.355,A -85,B 0,C 180,E1 18851.12,E2 18851.12} C_VEL
LIN {X 0,Y 419.162,Z 995.799,A -85,B 0,C 180,E1 18850.093,E2 18850.093} C_VEL
LIN {X 0,Y 416.272,Z 1015.18,A -85,B 0,C 180,E1 18848.821,E2 18848.821} C_VEL
LIN {X 0,Y 413.183,Z 1033.131,A -85,B 0,C 180,E1 18847.4,E2 18847.4} C_VEL
LIN {X 0,Y 409.621,Z 1050.99,A -85,B 0,C 180,E1 18845.688,E2 18845.688} C_VEL
LIN {X 0,Y 405.919,Z 1068.029,A -85,B 0,C 180,E1 18843.741,E2 18843.741} C_VEL
LIN {X 0,Y 402.303,Z 1083.691,A -85,B 0,C 180,E1 18841.627,E2 18841.627} C_VEL
LIN {X 0,Y 398.625,Z 1098.723,A -85,B 0,C 180,E1 18839.205,E2 18839.205} C_VEL
LIN {X 0,Y 395.317,Z 1111.962,A -85,B 0,C 180,E1 18836.669,E2 18836.669} C_VEL
LIN {X 0,Y 392.354,Z 1124.138,A -85,B 0,C 180,E1 18833.902,E2 18833.902} C_VEL
LIN {X 0,Y 390.976,Z 1129.934,A -85,B 0,C 180,E1 18832.392,E2 18832.392} C_VEL
LIN {X 0,Y 389.191,Z 1133.699,A -85,B 0,C 180,E1 18831.421,E2 18831.421} C_VEL
LIN {X 0,Y 381.662,Z 1143.134,A -85,B 0,C 180,E1 18829.023,E2 18829.023} C_VEL
LIN {X 0,Y 380.108,Z 1146.223,A -85,B 0,C 180,E1 18827.984,E2 18827.984} C_VEL
LIN {X 0,Y 378.645,Z 1153.502,A -85,B 0,C 180,E1 18824.841,E2 18824.841} C_VEL
LIN {X 0,Y 377.65,Z 1159.435,A -85,B 0,C 180,E1 18821.59,E2 18821.59} C_VEL
LIN {X 0,Y 377.094,Z 1163.71,A -85,B 0,C 180,E1 18818.385,E2 18818.385} C_VEL
LIN {X 0,Y 376.766,Z 1166.675,A -85,B 0,C 180,E1 18815.024,E2 18815.024} C_VEL
LIN {X 0,Y 376.661,Z 1168.178,A -85,B 0,C 180,E1 18811.825,E2 18811.825} C_VEL
LIN {X 0,Y 376.661,Z 1168.244,A -85,B 0,C 180,E1 18808.631,E2 18808.631} C_VEL
LIN {X 0,Y 376.756,Z 1166.937,A -85,B 0,C 180,E1 18805.281,E2 18805.281} C_VEL
LIN {X 0,Y 377.029,Z 1164.345,A -85,B 0,C 180,E1 18802.074,E2 18802.074} C_VEL
LIN {X 0,Y 377.522,Z 1160.222,A -85,B 0,C 180,E1 18798.853,E2 18798.853} C_VEL
LIN {X 0,Y 378.494,Z 1154.328,A -85,B 0,C 180,E1 18795.466,E2 18795.466} C_VEL
LIN {X 0,Y 379.959,Z 1147.044,A -85,B 0,C 180,E1 18792.227,E2 18792.227} C_VEL
LIN {X 0,Y 382.056,Z 1137.798,A -85,B 0,C 180,E1 18788.99,E2 18788.99} C_VEL
LIN {X 0,Y 384.542,Z 1127.639,A -85,B 0,C 180,E1 18786.071,E2 18786.071} C_VEL
LIN {X 0,Y 387.502,Z 1116.259,A -85,B 0,C 180,E1 18783.324,E2 18783.324} C_VEL
LIN {X 0,Y 390.894,Z 1103.337,A -85,B 0,C 180,E1 18780.72,E2 18780.72} C_VEL
LIN {X 0,Y 394.571,Z 1088.971,A -85,B 0,C 180,E1 18778.278,E2 18778.278} C_VEL
LIN {X 0,Y 398.423,Z 1073.532,A -85,B 0,C 180,E1 18776.058,E2 18776.058} C_VEL
LIN {X 0,Y 402.224,Z 1057.176,A -85,B 0,C 180,E1 18774.081,E2 18774.081} C_VEL
LIN {X 0,Y 405.998,Z 1039.182,A -85,B 0,C 180,E1 18772.259,E2 18772.259} C_VEL
LIN {X 0,Y 409.501,Z 1020.62,A -85,B 0,C 180,E1 18770.694,E2 18770.694} C_VEL
LIN {X 0,Y 412.514,Z 1001.973,A -85,B 0,C 180,E1 18769.4,E2 18769.4} C_VEL
LIN {X 0,Y 415.078,Z 982.519,A -85,B 0,C 180,E1 18768.309,E2 18768.309} C_VEL
LIN {X 0,Y 417.201,Z 962.215,A -85,B 0,C 180,E1 18767.407,E2 18767.407} C_VEL
LIN {X 0,Y 418.675,Z 941.178,A -85,B 0,C 180,E1 18766.717,E2 18766.717} C_VEL
LIN {X 0,Y 419.842,Z 912.768,A -85,B 0,C 180,E1 18766.103,E2 18766.103} C_VEL
LIN {X 0,Y 425.997,Z 754.296,A -85,B 0,C 180,E1 18763.148,E2 18763.148} C_VEL
LIN {X 0,Y 415.358,Z 738.113,A -85,B 0,C 180,E1 18761.062,E2 18761.062} C_VEL
LIN {X 0,Y 406.014,Z 724.87,A -85,B 0,C 180,E1 18759.082,E2 18759.082} C_VEL
LIN {X 0,Y 398.408,Z 714.802,A -85,B 0,C 180,E1 18757.352,E2 18757.352} C_VEL
LIN {X 0,Y 394.787,Z 710.067,A -85,B 0,C 180,E1 18756.48,E2 18756.48} C_VEL
LIN {X 0,Y 390.868,Z 705.018,A -85,B 0,C 180,E1 18755.498,E2 18755.498} C_VEL
LIN {X 0,Y 387.653,Z 700.971,A -85,B 0,C 180,E1 18754.662,E2 18754.662} C_VEL
LIN {X 0,Y 386.685,Z 699.682,A -85,B 0,C 180,E1 18754.401,E2 18754.401} C_VEL
LIN {X 0,Y 383.746,Z 696.627,A -85,B 0,C 180,E1 18753.62,E2 18753.62} C_VEL
LIN {X 0,Y 382.159,Z 693.922,A -85,B 0,C 180,E1 18753.149,E2 18753.149} C_VEL
LIN {X 0,Y 379.155,Z 691.378,A -85,B 0,C 180,E1 18752.322,E2 18752.322} C_VEL
LIN {X 0,Y 377.812,Z 688.398,A -85,B 0,C 180,E1 18751.779,E2 18751.779} C_VEL
LIN {X 0,Y 377.68,Z 687.666,A -85,B 0,C 180,E1 18751.258,E2 18751.258} C_VEL
LIN {X 0,Y 377.682,Z 687.662,A -85,B 0,C 180,E1 18747.192,E2 18747.192} C_VEL
LIN {X 0,Y 377.689,Z 687.677,A -85,B 0,C 180,E1 18743.067,E2 18743.067} C_VEL
LIN {X 0,Y 377.682,Z 687.677,A -85,B 0,C 180,E1 18739.004,E2 18739.004} C_VEL
LIN {X 0,Y 377.678,Z 687.673,A -85,B 0,C 180,E1 18734.88,E2 18734.88} C_VEL
LIN {X 0,Y 377.674,Z 687.667,A -85,B 0,C 180,E1 18730.834,E2 18730.834} C_VEL
LIN {X 0,Y 377.682,Z 687.662,A -85,B 0,C 180,E1 18726.842,E2 18726.842} C_VEL
LIN {X 0,Y 377.679,Z 687.667,A -85,B 0,C 180,E1 18722.732,E2 18722.732} C_VEL
LIN {X 0,Y 377.682,Z 687.678,A -85,B 0,C 180,E1 18718.635,E2 18718.635} C_VEL
LIN {X 0,Y 377.681,Z 687.688,A -85,B 0,C 180,E1 18714.488,E2 18714.488} C_VEL
LIN {X 0,Y 377.681,Z 687.691,A -85,B 0,C 180,E1 18710.399,E2 18710.399} C_VEL
LIN {X 0,Y 377.679,Z 687.64,A -85,B 0,C 180,E1 18706.302,E2 18706.302} C_VEL
LIN {X 0,Y 377.678,Z 687.655,A -85,B 0,C 180,E1 18702.275,E2 18702.275} C_VEL
LIN {X 0,Y 377.679,Z 687.69,A -85,B 0,C 180,E1 18698.246,E2 18698.246} C_VEL
LIN {X 0,Y 377.695,Z 687.813,A -85,B 0,C 180,E1 18694.269,E2 18694.269} C_VEL
LIN {X 0,Y 377.855,Z 688.624,A -85,B 0,C 180,E1 18693.944,E2 18693.944} C_VEL
LIN {X 0,Y 379.757,Z 692.153,A -85,B 0,C 180,E1 18692.904,E2 18692.904} C_VEL
LIN {X 0,Y 380.69,Z 693.583,A -85,B 0,C 180,E1 18692.468,E2 18692.468} C_VEL
LIN {X 0,Y 382.767,Z 697.304,A -85,B 0,C 180,E1 18691.444,E2 18691.444} C_VEL
LIN {X 0,Y 386.409,Z 704.108,A -85,B 0,C 180,E1 18689.697,E2 18689.697} C_VEL
LIN {X 0,Y 391.227,Z 713.131,A -85,B 0,C 180,E1 18687.541,E2 18687.541} C_VEL
LIN {X 0,Y 397.365,Z 725.202,A -85,B 0,C 180,E1 18684.992,E2 18684.992} C_VEL
LIN {X 0,Y 407.982,Z 742.009,A -85,B 0,C 180,E1 18682.527,E2 18682.527} C_VEL
LIN {X 0,Y 418.138,Z 759.522,A -85,B 0,C 180,E1 18680.368,E2 18680.368} C_VEL
LIN {X 0,Y 422.149,Z 767.286,A -85,B 0,C 180,E1 18679.548,E2 18679.548} C_VEL
LIN {X 0,Y 425.824,Z 802.207,A -85,B 0,C 180,E1 18678.144,E2 18678.144} C_VEL
LIN {X 0,Y 417.448,Z 1027.961,A -85,B 0,C 180,E1 18673.964,E2 18673.964} C_VEL
LIN {X 0,Y 416.087,Z 1051.968,A -85,B 0,C 180,E1 18673.44,E2 18673.44} C_VEL
LIN {X 0,Y 413.682,Z 1074.873,A -85,B 0,C 180,E1 18672.745,E2 18672.745} C_VEL
LIN {X 0,Y 410.783,Z 1096.114,A -85,B 0,C 180,E1 18671.871,E2 18671.871} C_VEL
LIN {X 0,Y 407.414,Z 1116.83,A -85,B 0,C 180,E1 18670.752,E2 18670.752} C_VEL
LIN {X 0,Y 403.49,Z 1138.595,A -85,B 0,C 180,E1 18669.28,E2 18669.28} C_VEL
LIN {X 0,Y 399.606,Z 1158.593,A -85,B 0,C 180,E1 18667.625,E2 18667.625} C_VEL
LIN {X 0,Y 395.661,Z 1177.709,A -85,B 0,C 180,E1 18665.713,E2 18665.713} C_VEL
LIN {X 0,Y 391.812,Z 1196.032,A -85,B 0,C 180,E1 18663.536,E2 18663.536} C_VEL
LIN {X 0,Y 388.269,Z 1213.01,A -85,B 0,C 180,E1 18661.171,E2 18661.171} C_VEL
LIN {X 0,Y 385.061,Z 1229.085,A -85,B 0,C 180,E1 18658.539,E2 18658.539} C_VEL
LIN {X 0,Y 382.33,Z 1243.656,A -85,B 0,C 180,E1 18655.728,E2 18655.728} C_VEL
LIN {X 0,Y 380.017,Z 1257.621,A -85,B 0,C 180,E1 18652.556,E2 18652.556} C_VEL
LIN {X 0,Y 378.499,Z 1268.653,A -85,B 0,C 180,E1 18649.602,E2 18649.602} C_VEL
LIN {X 0,Y 377.442,Z 1278.33,A -85,B 0,C 180,E1 18646.465,E2 18646.465} C_VEL
LIN {X 0,Y 376.809,Z 1286.688,A -85,B 0,C 180,E1 18643.138,E2 18643.138} C_VEL
LIN {X 0,Y 376.564,Z 1292.723,A -85,B 0,C 180,E1 18640.093,E2 18640.093} C_VEL
LIN {X 0,Y 376.524,Z 1297.108,A -85,B 0,C 180,E1 18637.016,E2 18637.016} C_VEL
LIN {X 0,Y 376.548,Z 1300.011,A -85,B 0,C 180,E1 18633.959,E2 18633.959} C_VEL
LIN {X 0,Y 376.599,Z 1301.181,A -85,B 0,C 180,E1 18631.065,E2 18631.065} C_VEL
LIN {X 0,Y 376.585,Z 1301.042,A -85,B 0,C 180,E1 18628.174,E2 18628.174} C_VEL
LIN {X 0,Y 376.551,Z 1299.261,A -85,B 0,C 180,E1 18625.126,E2 18625.126} C_VEL
LIN {X 0,Y 376.505,Z 1296.004,A -85,B 0,C 180,E1 18622.063,E2 18622.063} C_VEL
LIN {X 0,Y 376.615,Z 1291.011,A -85,B 0,C 180,E1 18618.98,E2 18618.98} C_VEL
LIN {X 0,Y 376.946,Z 1284.462,A -85,B 0,C 180,E1 18615.876,E2 18615.876} C_VEL
LIN {X 0,Y 377.659,Z 1276.078,A -85,B 0,C 180,E1 18612.752,E2 18612.752} C_VEL
LIN {X 0,Y 378.903,Z 1265.502,A -85,B 0,C 180,E1 18609.517,E2 18609.517} C_VEL
LIN {X 0,Y 380.648,Z 1253.633,A -85,B 0,C 180,E1 18606.469,E2 18606.469} C_VEL
LIN {X 0,Y 382.925,Z 1240.331,A -85,B 0,C 180,E1 18603.586,E2 18603.586} C_VEL
LIN {X 0,Y 385.758,Z 1225.451,A -85,B 0,C 180,E1 18600.839,E2 18600.839} C_VEL
LIN {X 0,Y 389.04,Z 1209.338,A -85,B 0,C 180,E1 18598.286,E2 18598.286} C_VEL
LIN {X 0,Y 392.683,Z 1191.903,A -85,B 0,C 180,E1 18595.934,E2 18595.934} C_VEL
LIN {X 0,Y 396.525,Z 1173.483,A -85,B 0,C 180,E1 18593.841,E2 18593.841} C_VEL
LIN {X 0,Y 400.577,Z 1153.593,A -85,B 0,C 180,E1 18591.939,E2 18591.939} C_VEL
LIN {X 0,Y 404.392,Z 1133.875,A -85,B 0,C 180,E1 18590.366,E2 18590.366} C_VEL
LIN {X 0,Y 408.013,Z 1113.283,A -85,B 0,C 180,E1 18589.042,E2 18589.042} C_VEL
LIN {X 0,Y 411.407,Z 1091.506,A -85,B 0,C 180,E1 18587.927,E2 18587.927} C_VEL
LIN {X 0,Y 414.237,Z 1070.286,A -85,B 0,C 180,E1 18587.094,E2 18587.094} C_VEL
LIN {X 0,Y 416.402,Z 1047.748,A -85,B 0,C 180,E1 18586.456,E2 18586.456} C_VEL
LIN {X 0,Y 417.882,Z 1015.009,A -85,B 0,C 180,E1 18585.802,E2 18585.802} C_VEL
LIN {X 0,Y 425.801,Z 800.711,A -85,B 0,C 180,E1 18581.827,E2 18581.827} C_VEL
LIN {X 0,Y 421.891,Z 766.472,A -85,B 0,C 180,E1 18580.404,E2 18580.404} C_VEL
LIN {X 0,Y 411.799,Z 748.443,A -85,B 0,C 180,E1 18578.32,E2 18578.32} C_VEL
LIN {X 0,Y 401.01,Z 730.989,A -85,B 0,C 180,E1 18575.913,E2 18575.913} C_VEL
LIN {X 0,Y 396.897,Z 724.322,A -85,B 0,C 180,E1 18574.879,E2 18574.879} C_VEL
LIN {X 0,Y 390.226,Z 711.133,A -85,B 0,C 180,E1 18572.031,E2 18572.031} C_VEL
LIN {X 0,Y 385.119,Z 701.703,A -85,B 0,C 180,E1 18569.727,E2 18569.727} C_VEL
LIN {X 0,Y 382.704,Z 697.231,A -85,B 0,C 180,E1 18568.562,E2 18568.562} C_VEL
LIN {X 0,Y 380.646,Z 693.46,A -85,B 0,C 180,E1 18567.536,E2 18567.536} C_VEL
LIN {X 0,Y 377.988,Z 689.089,A -85,B 0,C 180,E1 18566.215,E2 18566.215} C_VEL
LIN {X 0,Y 377.701,Z 687.854,A -85,B 0,C 180,E1 18565.838,E2 18565.838} C_VEL
LIN {X 0,Y 377.684,Z 687.692,A -85,B 0,C 180,E1 18561.917,E2 18561.917} C_VEL
LIN {X 0,Y 377.678,Z 687.652,A -85,B 0,C 180,E1 18557.884,E2 18557.884} C_VEL
LIN {X 0,Y 377.671,Z 687.644,A -85,B 0,C 180,E1 18553.94,E2 18553.94} C_VEL
LIN {X 0,Y 377.679,Z 687.692,A -85,B 0,C 180,E1 18549.755,E2 18549.755} C_VEL
LIN {X 0,Y 377.681,Z 687.687,A -85,B 0,C 180,E1 18545.621,E2 18545.621} C_VEL
LIN {X 0,Y 377.679,Z 687.675,A -85,B 0,C 180,E1 18541.517,E2 18541.517} C_VEL
LIN {X 0,Y 377.677,Z 687.665,A -85,B 0,C 180,E1 18537.42,E2 18537.42} C_VEL
LIN {X 0,Y 377.679,Z 687.663,A -85,B 0,C 180,E1 18533.31,E2 18533.31} C_VEL
LIN {X 0,Y 377.675,Z 687.667,A -85,B 0,C 180,E1 18529.16,E2 18529.16} C_VEL
LIN {X 0,Y 377.677,Z 687.674,A -85,B 0,C 180,E1 18525.076,E2 18525.076} C_VEL
LIN {X 0,Y 377.681,Z 687.676,A -85,B 0,C 180,E1 18520.923,E2 18520.923} C_VEL
LIN {X 0,Y 377.686,Z 687.676,A -85,B 0,C 180,E1 18516.768,E2 18516.768} C_VEL
LIN {X 0,Y 377.685,Z 687.662,A -85,B 0,C 180,E1 18512.742,E2 18512.742} C_VEL
LIN {X 0,Y 377.68,Z 687.635,A -85,B 0,C 180,E1 18508.742,E2 18508.742} C_VEL
LIN {X 0,Y 377.758,Z 688.14,A -85,B 0,C 180,E1 18508.169,E2 18508.169} C_VEL
LIN {X 0,Y 378.465,Z 690.245,A -85,B 0,C 180,E1 18507.769,E2 18507.769} C_VEL
LIN {X 0,Y 380.592,Z 692.89,A -85,B 0,C 180,E1 18507.146,E2 18507.146} C_VEL
LIN {X 0,Y 382.55,Z 694.385,A -85,B 0,C 180,E1 18506.621,E2 18506.621} C_VEL
LIN {X 0,Y 384.857,Z 698.068,A -85,B 0,C 180,E1 18505.953,E2 18505.953} C_VEL
LIN {X 0,Y 387.407,Z 700.535,A -85,B 0,C 180,E1 18505.291,E2 18505.291} C_VEL
LIN {X 0,Y 390.539,Z 704.717,A -85,B 0,C 180,E1 18504.467,E2 18504.467} C_VEL
LIN {X 0,Y 392.184,Z 706.665,A -85,B 0,C 180,E1 18504.054,E2 18504.054} C_VEL
LIN {X 0,Y 396.915,Z 712.85,A -85,B 0,C 180,E1 18502.892,E2 18502.892} C_VEL
LIN {X 0,Y 404.473,Z 722.791,A -85,B 0,C 180,E1 18501.151,E2 18501.151} C_VEL
LIN {X 0,Y 414.356,Z 736.671,A -85,B 0,C 180,E1 18499.039,E2 18499.039} C_VEL
LIN {X 0,Y 425.166,Z 753.007,A -85,B 0,C 180,E1 18496.908,E2 18496.908} C_VEL
LIN {X 0,Y 426.041,Z 754.816,A -85,B 0,C 180,E1 18496.732,E2 18496.732} C_VEL
LIN {X 0,Y 418.956,Z 935.127,A -85,B 0,C 180,E1 18493.347,E2 18493.347} C_VEL
LIN {X 0,Y 417.554,Z 956.991,A -85,B 0,C 180,E1 18492.691,E2 18492.691} C_VEL
LIN {X 0,Y 415.607,Z 977.756,A -85,B 0,C 180,E1 18491.835,E2 18491.835} C_VEL
LIN {X 0,Y 413.167,Z 997.198,A -85,B 0,C 180,E1 18490.797,E2 18490.797} C_VEL
LIN {X 0,Y 410.163,Z 1016.577,A -85,B 0,C 180,E1 18489.511,E2 18489.511} C_VEL
LIN {X 0,Y 406.948,Z 1034.528,A -85,B 0,C 180,E1 18488.074,E2 18488.074} C_VEL
LIN {X 0,Y 403.234,Z 1052.389,A -85,B 0,C 180,E1 18486.342,E2 18486.342} C_VEL
LIN {X 0,Y 399.365,Z 1069.429,A -85,B 0,C 180,E1 18484.371,E2 18484.371} C_VEL
LIN {X 0,Y 395.579,Z 1085.092,A -85,B 0,C 180,E1 18482.229,E2 18482.229} C_VEL
LIN {X 0,Y 391.747,Z 1099.979,A -85,B 0,C 180,E1 18479.798,E2 18479.798} C_VEL
LIN {X 0,Y 388.334,Z 1112.982,A -85,B 0,C 180,E1 18477.277,E2 18477.277} C_VEL
LIN {X 0,Y 385.25,Z 1124.959,A -85,B 0,C 180,E1 18474.535,E2 18474.535} C_VEL
LIN {X 0,Y 382.586,Z 1135.526,A -85,B 0,C 180,E1 18471.622,E2 18471.622} C_VEL
LIN {X 0,Y 380.423,Z 1144.715,A -85,B 0,C 180,E1 18468.543,E2 18468.543} C_VEL
LIN {X 0,Y 380.108,Z 1146.223,A -85,B 0,C 180,E1 18467.984,E2 18467.984} C_VEL
LIN {X 0,Y 378.607,Z 1149.208,A -85,B 0,C 180,E1 18466.925,E2 18466.925} C_VEL
LIN {X 0,Y 371.157,Z 1157.014,A -85,B 0,C 180,E1 18464.023,E2 18464.023} C_VEL
LIN {X 0,Y 370.221,Z 1158.705,A -85,B 0,C 180,E1 18463.127,E2 18463.127} C_VEL
LIN {X 0,Y 369.464,Z 1163.651,A -85,B 0,C 180,E1 18459.816,E2 18459.816} C_VEL
LIN {X 0,Y 369.023,Z 1167.054,A -85,B 0,C 180,E1 18456.534,E2 18456.534} C_VEL
LIN {X 0,Y 368.815,Z 1169.121,A -85,B 0,C 180,E1 18453.108,E2 18453.108} C_VEL
LIN {X 0,Y 368.782,Z 1169.797,A -85,B 0,C 180,E1 18449.845,E2 18449.845} C_VEL
LIN {X 0,Y 368.825,Z 1169.04,A -85,B 0,C 180,E1 18446.581,E2 18446.581} C_VEL
LIN {X 0,Y 369.062,Z 1166.719,A -85,B 0,C 180,E1 18442.998,E2 18442.998} C_VEL
LIN {X 0,Y 369.534,Z 1163.202,A -85,B 0,C 180,E1 18439.713,E2 18439.713} C_VEL
LIN {X 0,Y 370.409,Z 1157.807,A -85,B 0,C 180,E1 18436.259,E2 18436.259} C_VEL
LIN {X 0,Y 371.777,Z 1151.023,A -85,B 0,C 180,E1 18432.954,E2 18432.954} C_VEL
LIN {X 0,Y 373.684,Z 1142.962,A -85,B 0,C 180,E1 18429.809,E2 18429.809} C_VEL
LIN {X 0,Y 376.225,Z 1133.03,A -85,B 0,C 180,E1 18426.673,E2 18426.673} C_VEL
LIN {X 0,Y 379.298,Z 1121.635,A -85,B 0,C 180,E1 18423.714,E2 18423.714} C_VEL
LIN {X 0,Y 382.831,Z 1108.856,A -85,B 0,C 180,E1 18420.937,E2 18420.937} C_VEL
LIN {X 0,Y 386.749,Z 1094.651,A -85,B 0,C 180,E1 18418.345,E2 18418.345} C_VEL
LIN {X 0,Y 390.786,Z 1079.172,A -85,B 0,C 180,E1 18415.994,E2 18415.994} C_VEL
LIN {X 0,Y 394.931,Z 1062.386,A -85,B 0,C 180,E1 18413.852,E2 18413.852} C_VEL
LIN {X 0,Y 398.829,Z 1045.31,A -85,B 0,C 180,E1 18412.016,E2 18412.016} C_VEL
LIN {X 0,Y 402.441,Z 1027.285,A -85,B 0,C 180,E1 18410.404,E2 18410.404} C_VEL
LIN {X 0,Y 405.86,Z 1007.629,A -85,B 0,C 180,E1 18408.956,E2 18408.956} C_VEL
LIN {X 0,Y 408.752,Z 987.851,A -85,B 0,C 180,E1 18407.774,E2 18407.774} C_VEL
LIN {X 0,Y 411.019,Z 967.704,A -85,B 0,C 180,E1 18406.831,E2 18406.831} C_VEL
LIN {X 0,Y 412.74,Z 946.217,A -85,B 0,C 180,E1 18406.075,E2 18406.075} C_VEL
LIN {X 0,Y 413.778,Z 924.821,A -85,B 0,C 180,E1 18405.547,E2 18405.547} C_VEL
LIN {X 0,Y 420.526,Z 757.951,A -85,B 0,C 180,E1 18402.405,E2 18402.405} C_VEL
LIN {X 0,Y 409.17,Z 740.713,A -85,B 0,C 180,E1 18400.083,E2 18400.083} C_VEL
LIN {X 0,Y 399.308,Z 726.899,A -85,B 0,C 180,E1 18397.887,E2 18397.887} C_VEL
LIN {X 0,Y 391.422,Z 716.527,A -85,B 0,C 180,E1 18395.981,E2 18395.981} C_VEL
LIN {X 0,Y 387.555,Z 711.556,A -85,B 0,C 180,E1 18394.987,E2 18394.987} C_VEL
LIN {X 0,Y 383.548,Z 706.468,A -85,B 0,C 180,E1 18393.909,E2 18393.909} C_VEL
LIN {X 0,Y 380.325,Z 702.646,A -85,B 0,C 180,E1 18393.01,E2 18393.01} C_VEL
LIN {X 0,Y 379.08,Z 700.868,A -85,B 0,C 180,E1 18392.642,E2 18392.642} C_VEL
LIN {X 0,Y 376.052,Z 697.795,A -85,B 0,C 180,E1 18391.766,E2 18391.766} C_VEL
LIN {X 0,Y 374.336,Z 694.927,A -85,B 0,C 180,E1 18391.21,E2 18391.21} C_VEL
LIN {X 0,Y 371.274,Z 692.414,A -85,B 0,C 180,E1 18390.283,E2 18390.283} C_VEL
LIN {X 0,Y 369.865,Z 689.323,A -85,B 0,C 180,E1 18389.651,E2 18389.651} C_VEL
LIN {X 0,Y 369.745,Z 688.654,A -85,B 0,C 180,E1 18389.128,E2 18389.128} C_VEL
LIN {X 0,Y 369.743,Z 688.656,A -85,B 0,C 180,E1 18384.952,E2 18384.952} C_VEL
LIN {X 0,Y 369.749,Z 688.655,A -85,B 0,C 180,E1 18380.913,E2 18380.913} C_VEL
LIN {X 0,Y 369.744,Z 688.658,A -85,B 0,C 180,E1 18376.813,E2 18376.813} C_VEL
LIN {X 0,Y 369.738,Z 688.667,A -85,B 0,C 180,E1 18372.812,E2 18372.812} C_VEL
LIN {X 0,Y 369.74,Z 688.678,A -85,B 0,C 180,E1 18368.71,E2 18368.71} C_VEL
LIN {X 0,Y 369.741,Z 688.678,A -85,B 0,C 180,E1 18364.654,E2 18364.654} C_VEL
LIN {X 0,Y 369.746,Z 688.666,A -85,B 0,C 180,E1 18360.465,E2 18360.465} C_VEL
LIN {X 0,Y 369.739,Z 688.658,A -85,B 0,C 180,E1 18356.279,E2 18356.279} C_VEL
LIN {X 0,Y 369.736,Z 688.654,A -85,B 0,C 180,E1 18352.229,E2 18352.229} C_VEL
LIN {X 0,Y 369.735,Z 688.634,A -85,B 0,C 180,E1 18348.14,E2 18348.14} C_VEL
LIN {X 0,Y 369.742,Z 688.679,A -85,B 0,C 180,E1 18343.989,E2 18343.989} C_VEL
LIN {X 0,Y 369.738,Z 688.637,A -85,B 0,C 180,E1 18339.775,E2 18339.775} C_VEL
LIN {X 0,Y 369.777,Z 688.92,A -85,B 0,C 180,E1 18336.088,E2 18336.088} C_VEL
LIN {X 0,Y 371.26,Z 692.429,A -85,B 0,C 180,E1 18334.987,E2 18334.987} C_VEL
LIN {X 0,Y 372.796,Z 694.51,A -85,B 0,C 180,E1 18334.247,E2 18334.247} C_VEL
LIN {X 0,Y 374.699,Z 698.141,A -85,B 0,C 180,E1 18333.195,E2 18333.195} C_VEL
LIN {X 0,Y 375.877,Z 700.153,A -85,B 0,C 180,E1 18332.601,E2 18332.601} C_VEL
LIN {X 0,Y 378.567,Z 704.945,A -85,B 0,C 180,E1 18331.263,E2 18331.263} C_VEL
LIN {X 0,Y 383.48,Z 714.128,A -85,B 0,C 180,E1 18328.919,E2 18328.919} C_VEL
LIN {X 0,Y 387.956,Z 722.562,A -85,B 0,C 180,E1 18327.014,E2 18327.014} C_VEL
LIN {X 0,Y 397.196,Z 736.841,A -85,B 0,C 180,E1 18324.666,E2 18324.666} C_VEL
LIN {X 0,Y 407.677,Z 754.01,A -85,B 0,C 180,E1 18322.25,E2 18322.25} C_VEL
LIN {X 0,Y 417.025,Z 770.871,A -85,B 0,C 180,E1 18320.253,E2 18320.253} C_VEL
LIN {X 0,Y 420.327,Z 803.647,A -85,B 0,C 180,E1 18318.916,E2 18318.916} C_VEL
LIN {X 0,Y 411.562,Z 1028.869,A -85,B 0,C 180,E1 18314.704,E2 18314.704} C_VEL
LIN {X 0,Y 410.131,Z 1051.825,A -85,B 0,C 180,E1 18314.186,E2 18314.186} C_VEL
LIN {X 0,Y 407.521,Z 1075.161,A -85,B 0,C 180,E1 18313.457,E2 18313.457} C_VEL
LIN {X 0,Y 404.513,Z 1096.063,A -85,B 0,C 180,E1 18312.576,E2 18312.576} C_VEL
LIN {X 0,Y 401.014,Z 1116.545,A -85,B 0,C 180,E1 18311.449,E2 18311.449} C_VEL
LIN {X 0,Y 397.041,Z 1137.422,A -85,B 0,C 180,E1 18310.017,E2 18310.017} C_VEL
LIN {X 0,Y 393.033,Z 1157.125,A -85,B 0,C 180,E1 18308.368,E2 18308.368} C_VEL
LIN {X 0,Y 389.026,Z 1175.531,A -85,B 0,C 180,E1 18306.511,E2 18306.511} C_VEL
LIN {X 0,Y 384.936,Z 1193.958,A -85,B 0,C 180,E1 18304.307,E2 18304.307} C_VEL
LIN {X 0,Y 381.187,Z 1211.029,A -85,B 0,C 180,E1 18301.906,E2 18301.906} C_VEL
LIN {X 0,Y 377.844,Z 1226.689,A -85,B 0,C 180,E1 18299.31,E2 18299.31} C_VEL
LIN {X 0,Y 374.892,Z 1241.41,A -85,B 0,C 180,E1 18296.448,E2 18296.448} C_VEL
LIN {X 0,Y 372.499,Z 1254.907,A -85,B 0,C 180,E1 18293.366,E2 18293.366} C_VEL
LIN {X 0,Y 370.751,Z 1266.643,A -85,B 0,C 180,E1 18290.193,E2 18290.193} C_VEL
LIN {X 0,Y 369.597,Z 1276.427,A -85,B 0,C 180,E1 18286.987,E2 18286.987} C_VEL
LIN {X 0,Y 368.919,Z 1284.796,A -85,B 0,C 180,E1 18283.638,E2 18283.638} C_VEL
LIN {X 0,Y 368.652,Z 1290.731,A -85,B 0,C 180,E1 18280.628,E2 18280.628} C_VEL
LIN {X 0,Y 368.607,Z 1295.518,A -85,B 0,C 180,E1 18277.324,E2 18277.324} C_VEL
LIN {X 0,Y 368.659,Z 1298.378,A -85,B 0,C 180,E1 18274.355,E2 18274.355} C_VEL
LIN {X 0,Y 368.717,Z 1299.763,A -85,B 0,C 180,E1 18271.243,E2 18271.243} C_VEL
LIN {X 0,Y 368.711,Z 1299.708,A -85,B 0,C 180,E1 18268.446,E2 18268.446} C_VEL
LIN {X 0,Y 368.658,Z 1298.121,A -85,B 0,C 180,E1 18265.333,E2 18265.333} C_VEL
LIN {X 0,Y 368.604,Z 1295.148,A -85,B 0,C 180,E1 18262.362,E2 18262.362} C_VEL
LIN {X 0,Y 368.67,Z 1290.13,A -85,B 0,C 180,E1 18259.041,E2 18259.041} C_VEL
LIN {X 0,Y 368.967,Z 1283.935,A -85,B 0,C 180,E1 18255.962,E2 18255.962} C_VEL
LIN {X 0,Y 369.683,Z 1275.523,A -85,B 0,C 180,E1 18252.692,E2 18252.692} C_VEL
LIN {X 0,Y 370.975,Z 1264.943,A -85,B 0,C 180,E1 18249.325,E2 18249.325} C_VEL
LIN {X 0,Y 372.739,Z 1253.498,A -85,B 0,C 180,E1 18246.274,E2 18246.274} C_VEL
LIN {X 0,Y 375.195,Z 1239.822,A -85,B 0,C 180,E1 18243.219,E2 18243.219} C_VEL
LIN {X 0,Y 378.207,Z 1224.864,A -85,B 0,C 180,E1 18240.373,E2 18240.373} C_VEL
LIN {X 0,Y 381.607,Z 1209.161,A -85,B 0,C 180,E1 18237.811,E2 18237.811} C_VEL
LIN {X 0,Y 385.328,Z 1192.174,A -85,B 0,C 180,E1 18235.462,E2 18235.462} C_VEL
LIN {X 0,Y 389.477,Z 1173.399,A -85,B 0,C 180,E1 18233.264,E2 18233.264} C_VEL
LIN {X 0,Y 393.536,Z 1154.648,A -85,B 0,C 180,E1 18231.411,E2 18231.411} C_VEL
LIN {X 0,Y 397.471,Z 1135.222,A -85,B 0,C 180,E1 18229.818,E2 18229.818} C_VEL
LIN {X 0,Y 401.214,Z 1115.305,A -85,B 0,C 180,E1 18228.481,E2 18228.481} C_VEL
LIN {X 0,Y 404.738,Z 1094.498,A -85,B 0,C 180,E1 18227.353,E2 18227.353} C_VEL
LIN {X 0,Y 407.749,Z 1073.276,A -85,B 0,C 180,E1 18226.477,E2 18226.477} C_VEL
LIN {X 0,Y 410.219,Z 1050.44,A -85,B 0,C 180,E1 18225.783,E2 18225.783} C_VEL
LIN {X 0,Y 411.636,Z 1026.049,A -85,B 0,C 180,E1 18225.248,E2 18225.248} C_VEL
LIN {X 0,Y 420.331,Z 802.568,A -85,B 0,C 180,E1 18221.069,E2 18221.069} C_VEL
LIN {X 0,Y 416.81,Z 770.476,A -85,B 0,C 180,E1 18219.716,E2 18219.716} C_VEL
LIN {X 0,Y 406.539,Z 752.192,A -85,B 0,C 180,E1 18217.518,E2 18217.518} C_VEL
LIN {X 0,Y 396.169,Z 735.245,A -85,B 0,C 180,E1 18215.107,E2 18215.107} C_VEL
LIN {X 0,Y 387.362,Z 721.492,A -85,B 0,C 180,E1 18212.823,E2 18212.823} C_VEL
LIN {X 0,Y 381.823,Z 711.157,A -85,B 0,C 180,E1 18210.357,E2 18210.357} C_VEL
LIN {X 0,Y 379.675,Z 707.129,A -85,B 0,C 180,E1 18209.329,E2 18209.329} C_VEL
LIN {X 0,Y 377.611,Z 703.186,A -85,B 0,C 180,E1 18208.292,E2 18208.292} C_VEL
LIN {X 0,Y 374.969,Z 698.46,A -85,B 0,C 180,E1 18206.956,E2 18206.956} C_VEL
LIN {X 0,Y 372.963,Z 694.993,A -85,B 0,C 180,E1 18205.911,E2 18205.911} C_VEL
LIN {X 0,Y 372.152,Z 693.486,A -85,B 0,C 180,E1 18205.459,E2 18205.459} C_VEL
LIN {X 0,Y 370.153,Z 690.367,A -85,B 0,C 180,E1 18204.411,E2 18204.411} C_VEL
LIN {X 0,Y 369.771,Z 688.892,A -85,B 0,C 180,E1 18203.928,E2 18203.928} C_VEL
LIN {X 0,Y 369.739,Z 688.633,A -85,B 0,C 180,E1 18199.921,E2 18199.921} C_VEL
LIN {X 0,Y 369.746,Z 688.672,A -85,B 0,C 180,E1 18195.689,E2 18195.689} C_VEL
LIN {X 0,Y 369.736,Z 688.64,A -85,B 0,C 180,E1 18191.543,E2 18191.543} C_VEL
LIN {X 0,Y 369.737,Z 688.653,A -85,B 0,C 180,E1 18187.458,E2 18187.458} C_VEL
LIN {X 0,Y 369.738,Z 688.655,A -85,B 0,C 180,E1 18183.41,E2 18183.41} C_VEL
LIN {X 0,Y 369.743,Z 688.661,A -85,B 0,C 180,E1 18179.225,E2 18179.225} C_VEL
LIN {X 0,Y 369.741,Z 688.672,A -85,B 0,C 180,E1 18175.035,E2 18175.035} C_VEL
LIN {X 0,Y 369.742,Z 688.679,A -85,B 0,C 180,E1 18170.976,E2 18170.976} C_VEL
LIN {X 0,Y 369.742,Z 688.675,A -85,B 0,C 180,E1 18166.776,E2 18166.776} C_VEL
LIN {X 0,Y 369.739,Z 688.666,A -85,B 0,C 180,E1 18162.662,E2 18162.662} C_VEL
LIN {X 0,Y 369.738,Z 688.664,A -85,B 0,C 180,E1 18158.47,E2 18158.47} C_VEL
LIN {X 0,Y 369.74,Z 688.664,A -85,B 0,C 180,E1 18154.362,E2 18154.362} C_VEL
LIN {X 0,Y 369.778,Z 688.856,A -85,B 0,C 180,E1 18150.431,E2 18150.431} C_VEL
LIN {X 0,Y 370.142,Z 690.314,A -85,B 0,C 180,E1 18149.995,E2 18149.995} C_VEL
LIN {X 0,Y 371.938,Z 693.176,A -85,B 0,C 180,E1 18149.374,E2 18149.374} C_VEL
LIN {X 0,Y 374.803,Z 695.459,A -85,B 0,C 180,E1 18148.52,E2 18148.52} C_VEL
LIN {X 0,Y 377.091,Z 699.136,A -85,B 0,C 180,E1 18147.795,E2 18147.795} C_VEL
LIN {X 0,Y 379.755,Z 701.652,A -85,B 0,C 180,E1 18147.042,E2 18147.042} C_VEL
LIN {X 0,Y 382.727,Z 705.724,A -85,B 0,C 180,E1 18146.189,E2 18146.189} C_VEL
LIN {X 0,Y 384.561,Z 707.665,A -85,B 0,C 180,E1 18145.698,E2 18145.698} C_VEL
LIN {X 0,Y 388.116,Z 712.108,A -85,B 0,C 180,E1 18144.755,E2 18144.755} C_VEL
LIN {X 0,Y 397.408,Z 724.387,A -85,B 0,C 180,E1 18142.447,E2 18142.447} C_VEL
LIN {X 0,Y 407.348,Z 738.122,A -85,B 0,C 180,E1 18140.201,E2 18140.201} C_VEL
LIN {X 0,Y 418.767,Z 755.248,A -85,B 0,C 180,E1 18137.838,E2 18137.838} C_VEL
LIN {X 0,Y 420.565,Z 758.329,A -85,B 0,C 180,E1 18137.478,E2 18137.478} C_VEL
LIN {X 0,Y 413.254,Z 936.231,A -85,B 0,C 180,E1 18134.106,E2 18134.106} C_VEL
LIN {X 0,Y 411.81,Z 958.166,A -85,B 0,C 180,E1 18133.443,E2 18133.443} C_VEL
LIN {X 0,Y 409.77,Z 979.156,A -85,B 0,C 180,E1 18132.569,E2 18132.569} C_VEL
LIN {X 0,Y 407.197,Z 998.895,A -85,B 0,C 180,E1 18131.503,E2 18131.503} C_VEL
LIN {X 0,Y 404.116,Z 1017.974,A -85,B 0,C 180,E1 18130.221,E2 18130.221} C_VEL
LIN {X 0,Y 400.77,Z 1035.925,A -85,B 0,C 180,E1 18128.769,E2 18128.769} C_VEL
LIN {X 0,Y 396.86,Z 1053.977,A -85,B 0,C 180,E1 18126.998,E2 18126.998} C_VEL
LIN {X 0,Y 392.814,Z 1071.021,A -85,B 0,C 180,E1 18124.998,E2 18124.998} C_VEL
LIN {X 0,Y 388.9,Z 1086.494,A -85,B 0,C 180,E1 18122.851,E2 18122.851} C_VEL
LIN {X 0,Y 384.916,Z 1101.231,A -85,B 0,C 180,E1 18120.412,E2 18120.412} C_VEL
LIN {X 0,Y 381.285,Z 1114.388,A -85,B 0,C 180,E1 18117.824,E2 18117.824} C_VEL
LIN {X 0,Y 378.023,Z 1126.366,A -85,B 0,C 180,E1 18115.036,E2 18115.036} C_VEL
LIN {X 0,Y 375.192,Z 1136.934,A -85,B 0,C 180,E1 18112.07,E2 18112.07} C_VEL
LIN {X 0,Y 372.883,Z 1146.122,A -85,B 0,C 180,E1 18108.932,E2 18108.932} C_VEL
LIN {X 0,Y 371.166,Z 1153.956,A -85,B 0,C 180,E1 18105.627,E2 18105.627} C_VEL
LIN {X 0,Y 370.221,Z 1158.705,A -85,B 0,C 180,E1 18103.127,E2 18103.127} C_VEL
LIN {X 0,Y 368.924,Z 1160.849,A -85,B 0,C 180,E1 18101.986,E2 18101.986} C_VEL
LIN {X 0,Y 362.22,Z 1166.218,A -85,B 0,C 180,E1 18098.935,E2 18098.935} C_VEL
LIN {X 0,Y 361.314,Z 1167.372,A -85,B 0,C 180,E1 18097.902,E2 18097.902} C_VEL
LIN {X 0,Y 361.014,Z 1169.86,A -85,B 0,C 180,E1 18094.607,E2 18094.607} C_VEL
LIN {X 0,Y 360.906,Z 1171.05,A -85,B 0,C 180,E1 18091.111,E2 18091.111} C_VEL
LIN {X 0,Y 360.926,Z 1170.911,A -85,B 0,C 180,E1 18087.777,E2 18087.777} C_VEL
LIN {X 0,Y 361.061,Z 1169.326,A -85,B 0,C 180,E1 18084.438,E2 18084.438} C_VEL
LIN {X 0,Y 361.501,Z 1166.068,A -85,B 0,C 180,E1 18080.769,E2 18080.769} C_VEL
LIN {X 0,Y 362.235,Z 1161.644,A -85,B 0,C 180,E1 18077.405,E2 18077.405} C_VEL
LIN {X 0,Y 363.476,Z 1155.546,A -85,B 0,C 180,E1 18074.034,E2 18074.034} C_VEL
LIN {X 0,Y 365.305,Z 1147.771,A -85,B 0,C 180,E1 18070.66,E2 18070.66} C_VEL
LIN {X 0,Y 367.751,Z 1138.641,A -85,B 0,C 180,E1 18067.459,E2 18067.459} C_VEL
LIN {X 0,Y 370.735,Z 1128.102,A -85,B 0,C 180,E1 18064.437,E2 18064.437} C_VEL
LIN {X 0,Y 374.169,Z 1116.193,A -85,B 0,C 180,E1 18061.599,E2 18061.599} C_VEL
LIN {X 0,Y 378.005,Z 1103.012,A -85,B 0,C 180,E1 18058.951,E2 18058.951} C_VEL
LIN {X 0,Y 382.138,Z 1088.416,A -85,B 0,C 180,E1 18056.491,E2 18056.491} C_VEL
LIN {X 0,Y 386.272,Z 1072.853,A -85,B 0,C 180,E1 18054.29,E2 18054.29} C_VEL
LIN {X 0,Y 390.487,Z 1055.931,A -85,B 0,C 180,E1 18052.269,E2 18052.269} C_VEL
LIN {X 0,Y 394.492,Z 1038.139,A -85,B 0,C 180,E1 18050.495,E2 18050.495} C_VEL
LIN {X 0,Y 397.979,Z 1020.382,A -85,B 0,C 180,E1 18049.027,E2 18049.027} C_VEL
LIN {X 0,Y 401.226,Z 1001.285,A -85,B 0,C 180,E1 18047.715,E2 18047.715} C_VEL
LIN {X 0,Y 403.943,Z 981.303,A -85,B 0,C 180,E1 18046.618,E2 18046.618} C_VEL
LIN {X 0,Y 406.131,Z 959.877,A -85,B 0,C 180,E1 18045.708,E2 18045.708} C_VEL
LIN {X 0,Y 407.632,Z 938.108,A -85,B 0,C 180,E1 18045.036,E2 18045.036} C_VEL
LIN {X 0,Y 410.959,Z 859.11,A -85,B 0,C 180,E1 18043.497,E2 18043.497} C_VEL
LIN {X 0,Y 415.117,Z 761.712,A -85,B 0,C 180,E1 18041.642,E2 18041.642} C_VEL
LIN {X 0,Y 404.169,Z 745.063,A -85,B 0,C 180,E1 18039.318,E2 18039.318} C_VEL
LIN {X 0,Y 395.34,Z 732.645,A -85,B 0,C 180,E1 18037.281,E2 18037.281} C_VEL
LIN {X 0,Y 387.963,Z 722.82,A -85,B 0,C 180,E1 18035.442,E2 18035.442} C_VEL
LIN {X 0,Y 384.277,Z 718.052,A -85,B 0,C 180,E1 18034.466,E2 18034.466} C_VEL
LIN {X 0,Y 380.327,Z 713.067,A -85,B 0,C 180,E1 18033.375,E2 18033.375} C_VEL
LIN {X 0,Y 376.971,Z 708.688,A -85,B 0,C 180,E1 18032.397,E2 18032.397} C_VEL
LIN {X 0,Y 372.987,Z 704.205,A -85,B 0,C 180,E1 18031.201,E2 18031.201} C_VEL
LIN {X 0,Y 371.599,Z 702.067,A -85,B 0,C 180,E1 18030.746,E2 18030.746} C_VEL
LIN {X 0,Y 368.509,Z 699.157,A -85,B 0,C 180,E1 18029.771,E2 18029.771} C_VEL
LIN {X 0,Y 366.711,Z 696.065,A -85,B 0,C 180,E1 18029.124,E2 18029.124} C_VEL
LIN {X 0,Y 363.522,Z 693.66,A -85,B 0,C 180,E1 18028.056,E2 18028.056} C_VEL
LIN {X 0,Y 361.933,Z 690.381,A -85,B 0,C 180,E1 18027.296,E2 18027.296} C_VEL
LIN {X 0,Y 361.811,Z 689.697,A -85,B 0,C 180,E1 18026.773,E2 18026.773} C_VEL
LIN {X 0,Y 361.813,Z 689.663,A -85,B 0,C 180,E1 18022.59,E2 18022.59} C_VEL
LIN {X 0,Y 361.812,Z 689.664,A -85,B 0,C 180,E1 18018.363,E2 18018.363} C_VEL
LIN {X 0,Y 361.815,Z 689.663,A -85,B 0,C 180,E1 18014.084,E2 18014.084} C_VEL
LIN {X 0,Y 361.81,Z 689.655,A -85,B 0,C 180,E1 18009.866,E2 18009.866} C_VEL
LIN {X 0,Y 361.809,Z 689.645,A -85,B 0,C 180,E1 18005.71,E2 18005.71} C_VEL
LIN {X 0,Y 361.806,Z 689.639,A -85,B 0,C 180,E1 18001.584,E2 18001.584} C_VEL
LIN {X 0,Y 361.801,Z 689.641,A -85,B 0,C 180,E1 17997.466,E2 17997.466} C_VEL
LIN {X 0,Y 361.801,Z 689.645,A -85,B 0,C 180,E1 17993.335,E2 17993.335} C_VEL
LIN {X 0,Y 361.798,Z 689.645,A -85,B 0,C 180,E1 17989.169,E2 17989.169} C_VEL
LIN {X 0,Y 361.797,Z 689.639,A -85,B 0,C 180,E1 17984.943,E2 17984.943} C_VEL
LIN {X 0,Y 361.794,Z 689.617,A -85,B 0,C 180,E1 17980.8,E2 17980.8} C_VEL
LIN {X 0,Y 361.845,Z 689.955,A -85,B 0,C 180,E1 17978.189,E2 17978.189} C_VEL
LIN {X 0,Y 363.358,Z 693.474,A -85,B 0,C 180,E1 17977,E2 17977} C_VEL
LIN {X 0,Y 364.878,Z 695.301,A -85,B 0,C 180,E1 17976.236,E2 17976.236} C_VEL
LIN {X 0,Y 366.88,Z 699.204,A -85,B 0,C 180,E1 17975.013,E2 17975.013} C_VEL
LIN {X 0,Y 368.02,Z 701.035,A -85,B 0,C 180,E1 17974.407,E2 17974.407} C_VEL
LIN {X 0,Y 370.98,Z 706.445,A -85,B 0,C 180,E1 17972.796,E2 17972.796} C_VEL
LIN {X 0,Y 373.894,Z 711.811,A -85,B 0,C 180,E1 17971.295,E2 17971.295} C_VEL
LIN {X 0,Y 378.194,Z 719.404,A -85,B 0,C 180,E1 17969.364,E2 17969.364} C_VEL
LIN {X 0,Y 387.033,Z 732.666,A -85,B 0,C 180,E1 17966.881,E2 17966.881} C_VEL
LIN {X 0,Y 397.067,Z 748.598,A -85,B 0,C 180,E1 17964.343,E2 17964.343} C_VEL
LIN {X 0,Y 407.349,Z 766.343,A -85,B 0,C 180,E1 17961.969,E2 17961.969} C_VEL
LIN {X 0,Y 412.058,Z 775.433,A -85,B 0,C 180,E1 17960.934,E2 17960.934} C_VEL
LIN {X 0,Y 414.914,Z 804.974,A -85,B 0,C 180,E1 17959.71,E2 17959.71} C_VEL
LIN {X 0,Y 405.742,Z 1029.672,A -85,B 0,C 180,E1 17955.467,E2 17955.467} C_VEL
LIN {X 0,Y 404.189,Z 1052.362,A -85,B 0,C 180,E1 17954.936,E2 17954.936} C_VEL
LIN {X 0,Y 401.523,Z 1074.726,A -85,B 0,C 180,E1 17954.217,E2 17954.217} C_VEL
LIN {X 0,Y 398.426,Z 1095.232,A -85,B 0,C 180,E1 17953.341,E2 17953.341} C_VEL
LIN {X 0,Y 394.945,Z 1114.786,A -85,B 0,C 180,E1 17952.258,E2 17952.258} C_VEL
LIN {X 0,Y 390.79,Z 1135.676,A -85,B 0,C 180,E1 17950.82,E2 17950.82} C_VEL
LIN {X 0,Y 386.525,Z 1155.656,A -85,B 0,C 180,E1 17949.136,E2 17949.136} C_VEL
LIN {X 0,Y 382.263,Z 1174.295,A -85,B 0,C 180,E1 17947.232,E2 17947.232} C_VEL
LIN {X 0,Y 378.003,Z 1192.474,A -85,B 0,C 180,E1 17945.028,E2 17945.028} C_VEL
LIN {X 0,Y 374.053,Z 1209.542,A -85,B 0,C 180,E1 17942.588,E2 17942.588} C_VEL
LIN {X 0,Y 370.489,Z 1225.198,A -85,B 0,C 180,E1 17939.951,E2 17939.951} C_VEL
LIN {X 0,Y 367.358,Z 1239.923,A -85,B 0,C 180,E1 17937.034,E2 17937.034} C_VEL
LIN {X 0,Y 364.834,Z 1253.276,A -85,B 0,C 180,E1 17933.928,E2 17933.928} C_VEL
LIN {X 0,Y 363.02,Z 1264.607,A -85,B 0,C 180,E1 17930.811,E2 17930.811} C_VEL
LIN {X 0,Y 361.751,Z 1274.524,A -85,B 0,C 180,E1 17927.531,E2 17927.531} C_VEL
LIN {X 0,Y 361.027,Z 1282.749,A -85,B 0,C 180,E1 17924.231,E2 17924.231} C_VEL
LIN {X 0,Y 360.74,Z 1288.823,A -85,B 0,C 180,E1 17921.137,E2 17921.137} C_VEL
LIN {X 0,Y 360.686,Z 1293.742,A -85,B 0,C 180,E1 17917.807,E2 17917.807} C_VEL
LIN {X 0,Y 360.764,Z 1296.725,A -85,B 0,C 180,E1 17914.769,E2 17914.769} C_VEL
LIN {X 0,Y 360.831,Z 1298.317,A -85,B 0,C 180,E1 17911.588,E2 17911.588} C_VEL
LIN {X 0,Y 360.84,Z 1298.399,A -85,B 0,C 180,E1 17908.889,E2 17908.889} C_VEL
LIN {X 0,Y 360.766,Z 1297.106,A -85,B 0,C 180,E1 17905.709,E2 17905.709} C_VEL
LIN {X 0,Y 360.698,Z 1294.29,A -85,B 0,C 180,E1 17902.674,E2 17902.674} C_VEL
LIN {X 0,Y 360.71,Z 1289.879,A -85,B 0,C 180,E1 17899.459,E2 17899.459} C_VEL
LIN {X 0,Y 360.954,Z 1284.043,A -85,B 0,C 180,E1 17896.382,E2 17896.382} C_VEL
LIN {X 0,Y 361.624,Z 1275.872,A -85,B 0,C 180,E1 17892.958,E2 17892.958} C_VEL
LIN {X 0,Y 362.792,Z 1266.226,A -85,B 0,C 180,E1 17889.681,E2 17889.681} C_VEL
LIN {X 0,Y 364.503,Z 1255.161,A -85,B 0,C 180,E1 17886.563,E2 17886.563} C_VEL
LIN {X 0,Y 366.912,Z 1242.197,A -85,B 0,C 180,E1 17883.455,E2 17883.455} C_VEL
LIN {X 0,Y 369.995,Z 1227.539,A -85,B 0,C 180,E1 17880.476,E2 17880.476} C_VEL
LIN {X 0,Y 373.513,Z 1211.75,A -85,B 0,C 180,E1 17877.768,E2 17877.768} C_VEL
LIN {X 0,Y 377.685,Z 1193.798,A -85,B 0,C 180,E1 17875.152,E2 17875.152} C_VEL
LIN {X 0,Y 381.846,Z 1176.116,A -85,B 0,C 180,E1 17872.97,E2 17872.97} C_VEL
LIN {X 0,Y 385.955,Z 1158.06,A -85,B 0,C 180,E1 17871.101,E2 17871.101} C_VEL
LIN {X 0,Y 390.202,Z 1138.408,A -85,B 0,C 180,E1 17869.396,E2 17869.396} C_VEL
LIN {X 0,Y 394.245,Z 1118.487,A -85,B 0,C 180,E1 17867.97,E2 17867.97} C_VEL
LIN {X 0,Y 397.955,Z 1097.75,A -85,B 0,C 180,E1 17866.793,E2 17866.793} C_VEL
LIN {X 0,Y 401.379,Z 1075.583,A -85,B 0,C 180,E1 17865.819,E2 17865.819} C_VEL
LIN {X 0,Y 404.052,Z 1053.62,A -85,B 0,C 180,E1 17865.102,E2 17865.102} C_VEL
LIN {X 0,Y 405.632,Z 1031.059,A -85,B 0,C 180,E1 17864.568,E2 17864.568} C_VEL
LIN {X 0,Y 414.743,Z 807.878,A -85,B 0,C 180,E1 17860.351,E2 17860.351} C_VEL
LIN {X 0,Y 414.758,Z 802.388,A -85,B 0,C 180,E1 17860.213,E2 17860.213} C_VEL
LIN {X 0,Y 411.821,Z 774.696,A -85,B 0,C 180,E1 17859.022,E2 17859.022} C_VEL
LIN {X 0,Y 402.09,Z 757.141,A -85,B 0,C 180,E1 17856.863,E2 17856.863} C_VEL
LIN {X 0,Y 391.785,Z 740.09,A -85,B 0,C 180,E1 17854.377,E2 17854.377} C_VEL
LIN {X 0,Y 382.384,Z 725.738,A -85,B 0,C 180,E1 17851.883,E2 17851.883} C_VEL
LIN {X 0,Y 377.381,Z 718.197,A -85,B 0,C 180,E1 17850.401,E2 17850.401} C_VEL
LIN {X 0,Y 372.355,Z 708.895,A -85,B 0,C 180,E1 17847.943,E2 17847.943} C_VEL
LIN {X 0,Y 369.905,Z 704.437,A -85,B 0,C 180,E1 17846.66,E2 17846.66} C_VEL
LIN {X 0,Y 367.126,Z 699.497,A -85,B 0,C 180,E1 17845.142,E2 17845.142} C_VEL
LIN {X 0,Y 365.009,Z 695.716,A -85,B 0,C 180,E1 17843.917,E2 17843.917} C_VEL
LIN {X 0,Y 362.111,Z 691.067,A -85,B 0,C 180,E1 17842.227,E2 17842.227} C_VEL
LIN {X 0,Y 361.816,Z 689.775,A -85,B 0,C 180,E1 17841.734,E2 17841.734} C_VEL
LIN {X 0,Y 361.799,Z 689.633,A -85,B 0,C 180,E1 17837.56,E2 17837.56} C_VEL
LIN {X 0,Y 361.801,Z 689.612,A -85,B 0,C 180,E1 17833.409,E2 17833.409} C_VEL
LIN {X 0,Y 361.806,Z 689.661,A -85,B 0,C 180,E1 17829.223,E2 17829.223} C_VEL
LIN {X 0,Y 361.807,Z 689.669,A -85,B 0,C 180,E1 17825.073,E2 17825.073} C_VEL
LIN {X 0,Y 361.813,Z 689.664,A -85,B 0,C 180,E1 17820.791,E2 17820.791} C_VEL
LIN {X 0,Y 361.806,Z 689.652,A -85,B 0,C 180,E1 17816.589,E2 17816.589} C_VEL
LIN {X 0,Y 361.814,Z 689.643,A -85,B 0,C 180,E1 17812.377,E2 17812.377} C_VEL
LIN {X 0,Y 361.808,Z 689.641,A -85,B 0,C 180,E1 17808.2,E2 17808.2} C_VEL
LIN {X 0,Y 361.808,Z 689.64,A -85,B 0,C 180,E1 17804.085,E2 17804.085} C_VEL
LIN {X 0,Y 361.808,Z 689.641,A -85,B 0,C 180,E1 17799.96,E2 17799.96} C_VEL
LIN {X 0,Y 361.806,Z 689.642,A -85,B 0,C 180,E1 17795.774,E2 17795.774} C_VEL
LIN {X 0,Y 361.833,Z 689.824,A -85,B 0,C 180,E1 17792.843,E2 17792.843} C_VEL
LIN {X 0,Y 362.181,Z 691.255,A -85,B 0,C 180,E1 17792.343,E2 17792.343} C_VEL
LIN {X 0,Y 364.02,Z 694.206,A -85,B 0,C 180,E1 17791.629,E2 17791.629} C_VEL
LIN {X 0,Y 367.072,Z 696.542,A -85,B 0,C 180,E1 17790.617,E2 17790.617} C_VEL
LIN {X 0,Y 369.259,Z 700.092,A -85,B 0,C 180,E1 17789.848,E2 17789.848} C_VEL
LIN {X 0,Y 372.16,Z 702.774,A -85,B 0,C 180,E1 17788.947,E2 17788.947} C_VEL
LIN {X 0,Y 375.132,Z 706.885,A -85,B 0,C 180,E1 17788.012,E2 17788.012} C_VEL
LIN {X 0,Y 376.997,Z 708.76,A -85,B 0,C 180,E1 17787.471,E2 17787.471} C_VEL
LIN {X 0,Y 380.487,Z 713.224,A -85,B 0,C 180,E1 17786.461,E2 17786.461} C_VEL
LIN {X 0,Y 386.653,Z 721.124,A -85,B 0,C 180,E1 17784.784,E2 17784.784} C_VEL
LIN {X 0,Y 393.987,Z 730.79,A -85,B 0,C 180,E1 17782.934,E2 17782.934} C_VEL
LIN {X 0,Y 403.85,Z 744.627,A -85,B 0,C 180,E1 17780.645,E2 17780.645} C_VEL
LIN {X 0,Y 414.939,Z 761.486,A -85,B 0,C 180,E1 17778.289,E2 17778.289} C_VEL
LIN {X 0,Y 415.123,Z 762.74,A -85,B 0,C 180,E1 17778.227,E2 17778.227} C_VEL
LIN {X 0,Y 407.625,Z 937.387,A -85,B 0,C 180,E1 17774.886,E2 17774.886} C_VEL
LIN {X 0,Y 406.133,Z 959.415,A -85,B 0,C 180,E1 17774.214,E2 17774.214} C_VEL
LIN {X 0,Y 404.077,Z 979.981,A -85,B 0,C 180,E1 17773.354,E2 17773.354} C_VEL
LIN {X 0,Y 401.429,Z 999.602,A -85,B 0,C 180,E1 17772.289,E2 17772.289} C_VEL
LIN {X 0,Y 398.132,Z 1019.372,A -85,B 0,C 180,E1 17770.954,E2 17770.954} C_VEL
LIN {X 0,Y 394.654,Z 1037.322,A -85,B 0,C 180,E1 17769.486,E2 17769.486} C_VEL
LIN {X 0,Y 390.626,Z 1055.186,A -85,B 0,C 180,E1 17767.715,E2 17767.715} C_VEL
LIN {X 0,Y 386.289,Z 1072.697,A -85,B 0,C 180,E1 17765.634,E2 17765.634} C_VEL
LIN {X 0,Y 382.12,Z 1088.401,A -85,B 0,C 180,E1 17763.415,E2 17763.415} C_VEL
LIN {X 0,Y 377.883,Z 1103.402,A -85,B 0,C 180,E1 17760.884,E2 17760.884} C_VEL
LIN {X 0,Y 374.062,Z 1116.511,A -85,B 0,C 180,E1 17758.236,E2 17758.236} C_VEL
LIN {X 0,Y 370.469,Z 1128.945,A -85,B 0,C 180,E1 17755.24,E2 17755.24} C_VEL
LIN {X 0,Y 367.555,Z 1139.389,A -85,B 0,C 180,E1 17752.217,E2 17752.217} C_VEL
LIN {X 0,Y 365.152,Z 1148.362,A -85,B 0,C 180,E1 17749.016,E2 17749.016} C_VEL
LIN {X 0,Y 363.35,Z 1156.065,A -85,B 0,C 180,E1 17745.608,E2 17745.608} C_VEL
LIN {X 0,Y 362.156,Z 1162.064,A -85,B 0,C 180,E1 17742.219,E2 17742.219} C_VEL
LIN {X 0,Y 361.439,Z 1166.505,A -85,B 0,C 180,E1 17738.751,E2 17738.751} C_VEL
LIN {X 0,Y 361.314,Z 1167.372,A -85,B 0,C 180,E1 17737.902,E2 17737.902} C_VEL
LIN {X 0,Y 360.171,Z 1168.639,A -85,B 0,C 180,E1 17736.698,E2 17736.698} C_VEL
LIN {X 0,Y 353.822,Z 1171.704,A -85,B 0,C 180,E1 17733.473,E2 17733.473} C_VEL
LIN {X 0,Y 353.051,Z 1172.217,A -85,B 0,C 180,E1 17732.4,E2 17732.4} C_VEL
LIN {X 0,Y 353.025,Z 1172.473,A -85,B 0,C 180,E1 17729.026,E2 17729.026} C_VEL
LIN {X 0,Y 353.135,Z 1171.516,A -85,B 0,C 180,E1 17725.616,E2 17725.616} C_VEL
LIN {X 0,Y 353.428,Z 1169.089,A -85,B 0,C 180,E1 17722.196,E2 17722.196} C_VEL
LIN {X 0,Y 354.076,Z 1165.096,A -85,B 0,C 180,E1 17718.6,E2 17718.6} C_VEL
LIN {X 0,Y 355.188,Z 1159.796,A -85,B 0,C 180,E1 17715.158,E2 17715.158} C_VEL
LIN {X 0,Y 356.866,Z 1152.734,A -85,B 0,C 180,E1 17711.712,E2 17711.712} C_VEL
LIN {X 0,Y 359.289,Z 1143.89,A -85,B 0,C 180,E1 17708.278,E2 17708.278} C_VEL
LIN {X 0,Y 362.148,Z 1134.19,A -85,B 0,C 180,E1 17705.188,E2 17705.188} C_VEL
LIN {X 0,Y 365.7,Z 1122.494,A -85,B 0,C 180,E1 17702.127,E2 17702.127} C_VEL
LIN {X 0,Y 369.623,Z 1109.668,A -85,B 0,C 180,E1 17699.341,E2 17699.341} C_VEL
LIN {X 0,Y 373.995,Z 1095.069,A -85,B 0,C 180,E1 17696.676,E2 17696.676} C_VEL
LIN {X 0,Y 378.507,Z 1079.425,A -85,B 0,C 180,E1 17694.284,E2 17694.284} C_VEL
LIN {X 0,Y 382.776,Z 1063.256,A -85,B 0,C 180,E1 17692.228,E2 17692.228} C_VEL
LIN {X 0,Y 387.183,Z 1044.977,A -85,B 0,C 180,E1 17690.274,E2 17690.274} C_VEL
LIN {X 0,Y 391.149,Z 1026.613,A -85,B 0,C 180,E1 17688.642,E2 17688.642} C_VEL
LIN {X 0,Y 394.479,Z 1008.294,A -85,B 0,C 180,E1 17687.311,E2 17687.311} C_VEL
LIN {X 0,Y 397.595,Z 987.728,A -85,B 0,C 180,E1 17686.098,E2 17686.098} C_VEL
LIN {X 0,Y 400.003,Z 967.47,A -85,B 0,C 180,E1 17685.156,E2 17685.156} C_VEL
LIN {X 0,Y 401.68,Z 946.42,A -85,B 0,C 180,E1 17684.433,E2 17684.433} C_VEL
LIN {X 0,Y 402.958,Z 918.937,A -85,B 0,C 180,E1 17683.798,E2 17683.798} C_VEL
LIN {X 0,Y 409.788,Z 765.458,A -85,B 0,C 180,E1 17680.861,E2 17680.861} C_VEL
LIN {X 0,Y 398.448,Z 748.241,A -85,B 0,C 180,E1 17678.349,E2 17678.349} C_VEL
LIN {X 0,Y 389.015,Z 735.015,A -85,B 0,C 180,E1 17676.057,E2 17676.057} C_VEL
LIN {X 0,Y 381.275,Z 724.803,A -85,B 0,C 180,E1 17674.003,E2 17674.003} C_VEL
LIN {X 0,Y 377.381,Z 719.857,A -85,B 0,C 180,E1 17672.898,E2 17672.898} C_VEL
LIN {X 0,Y 373.16,Z 714.559,A -85,B 0,C 180,E1 17671.635,E2 17671.635} C_VEL
LIN {X 0,Y 369.751,Z 710.259,A -85,B 0,C 180,E1 17670.556,E2 17670.556} C_VEL
LIN {X 0,Y 368.668,Z 708.974,A -85,B 0,C 180,E1 17670.205,E2 17670.205} C_VEL
